  MoveL 668 to (230.14, 163.68, 22.22) mm, rotated rx 180 ry 0 rz -160 deg; joints [-25.106, 26.658, 31.364, 9.576, 32.341, -8.112]
  Call Extruder(552.80049)
  MoveL 669 to (229.91, 163.75, 22.22) mm, rotated rx 180 ry 0 rz -180 deg; joints [-30.703, 36.195, 15.324, 43.661, 47.695, -32.714]
  MoveL 670 to (229.91, 163.75, 22.22) mm, rotated rx -180 ry 0 rz 180 deg; joints [-30.703, 36.195, 15.324, 43.661, 47.695, -32.714]
  Call Extruder(553.06879)
  MoveL 671 to (229.69, 163.82, 22.23) mm, rotated rx 180 ry 0 rz 180 deg; joints [-30.721, 35.901, 15.858, 43.833, 47.531, -32.953]
  MoveL 672 to (229.69, 163.82, 22.23) mm, rotated rx 180 ry 0 rz 180 deg; joints [-30.721, 35.901, 15.858, 43.833, 47.531, -32.953]
  Call Extruder(553.30777)
  MoveL 673 to (229.48, 163.86, 22.23) mm, rotated rx 180 ry 0 rz 180 deg; joints [-30.736, 35.656, 16.302, 43.977, 47.396, -33.151]
  MoveL 674 to (229.48, 163.86, 22.23) mm, rotated rx 180 ry 0 rz 180 deg; joints [-30.736, 35.656, 16.302, 43.977, 47.396, -33.151]
  Call Extruder(553.54569)
  MoveL 675 to (229.28, 163.91, 22.22) mm, rotated rx 180 ry 0 rz 180 deg; joints [-30.751, 35.437, 16.698, 44.107, 47.277, -33.33]
  MoveL 676 to (229.28, 163.91, 22.22) mm, rotated rx 180 ry 0 rz 180 deg; joints [-30.751, 35.437, 16.698, 44.107, 47.277, -33.33]
  Call Extruder(553.78253)
  MoveL 677 to (229.08, 163.95, 22.23) mm, rotated rx 180 ry 0 rz 180 deg; joints [-30.766, 35.235, 17.061, 44.227, 47.17, -33.494]
  MoveL 678 to (229.08, 163.95, 22.23) mm, rotated rx 180 ry 0 rz 180 deg; joints [-30.766, 35.235, 17.061, 44.227, 47.17, -33.494]
  Call Extruder(554.01831)
  MoveL 679 to (228.87, 164, 22.23) mm, rotated rx 180 ry 0 rz 180 deg; joints [-30.781, 35.047, 17.397, 44.341, 47.072, -33.647]
  MoveL 680 to (228.87, 164, 22.23) mm, rotated rx 180 ry 0 rz 180 deg; joints [-30.781, 35.047, 17.397, 44.341, 47.072, -33.647]
  Call Extruder(554.27820)
  MoveL 681 to (228.64, 164.04, 22.23) mm, rotated rx -180 ry 0 rz -180 deg; joints [-30.797, 34.852, 17.746, 44.459, 46.971, -33.806]
  MoveL 682 to (228.64, 164.04, 22.23) mm, rotated rx -180 ry 0 rz -180 deg; joints [-30.797, 34.852, 17.746, 44.459, 46.971, -33.806]
  Call Extruder(554.56187)
  MoveL 683 to (228.4, 164.09, 22.22) mm, rotated rx 180 ry 0 rz -180 deg; joints [-30.815, 34.649, 18.106, 44.582, 46.869, -33.971]
  MoveL 684 to (228.4, 164.09, 22.22) mm, rotated rx 180 ry 0 rz -180 deg; joints [-30.815, 34.649, 18.106, 44.582, 46.869, -33.971]
  Call Extruder(554.84409)
  MoveL 685 to (228.15, 164.14, 22.22) mm, rotated rx 180 ry 0 rz 180 deg; joints [-30.832, 34.457, 18.446, 44.7, 46.773, -34.128]
  MoveL 686 to (228.15, 164.14, 22.22) mm, rotated rx 180 ry 0 rz 180 deg; joints [-30.832, 34.457, 18.446, 44.7, 46.773, -34.128]
  Call Extruder(555.12487)
  MoveL 687 to (227.9, 164.19, 22.23) mm, rotated rx 180 ry 0 rz 180 deg; joints [-30.85, 34.276, 18.766, 44.812, 46.685, -34.276]
  MoveL 688 to (227.9, 164.19, 22.23) mm, rotated rx 180 ry 0 rz 180 deg; joints [-30.85, 34.276, 18.766, 44.812, 46.685, -34.276]
  Call Extruder(555.40421)
  MoveL 689 to (227.65, 164.24, 22.22) mm, rotated rx 180 ry 0 rz 180 deg; joints [-30.868, 34.103, 19.07, 44.92, 46.602, -34.417]
  MoveL 690 to (227.65, 164.24, 22.22) mm, rotated rx 180 ry 0 rz 180 deg; joints [-30.868, 34.103, 19.07, 44.92, 46.602, -34.417]
  Call Extruder(555.68211)
  MoveL 691 to (227.4, 164.29, 22.23) mm, rotated rx -180 ry 0 rz -180 deg; joints [-30.886, 33.937, 19.361, 45.024, 46.523, -34.552]
  MoveL 692 to (227.4, 164.29, 22.23) mm, rotated rx -180 ry 0 rz -180 deg; joints [-30.886, 33.937, 19.361, 45.024, 46.523, -34.552]
  Call Extruder(555.95856)
  MoveL 693 to (227.15, 164.34, 22.22) mm, rotated rx 180 ry 0 rz 180 deg; joints [-30.903, 33.778, 19.639, 45.124, 46.449, -34.683]
  MoveL 694 to (227.15, 164.34, 22.22) mm, rotated rx 180 ry 0 rz 180 deg; joints [-30.903, 33.778, 19.639, 45.124, 46.449, -34.683]
  Call Extruder(556.26358)
  MoveL 695 to (226.87, 164.39, 22.23) mm, rotated rx 180 ry 0 rz 180 deg; joints [-30.923, 33.605, 19.941, 45.233, 46.369, -34.824]
  MoveL 696 to (226.87, 164.39, 22.23) mm, rotated rx 180 ry 0 rz 180 deg; joints [-30.923, 33.605, 19.941, 45.233, 46.369, -34.824]
  Call Extruder(556.59701)
  MoveL 697 to (226.57, 164.44, 22.22) mm, rotated rx 180 ry 0 rz 180 deg; joints [-30.943, 33.419, 20.264, 45.349, 46.284, -34.975]
  MoveL 698 to (226.57, 164.44, 22.22) mm, rotated rx 180 ry 0 rz 180 deg; joints [-30.943, 33.419, 20.264, 45.349, 46.284, -34.975]
  Call Extruder(556.92871)
  MoveL 699 to (226.26, 164.49, 22.22) mm, rotated rx -180 ry 0 rz 180 deg; joints [-30.964, 33.24, 20.575, 45.463, 46.204, -35.121]
  MoveL 700 to (226.26, 164.49, 22.22) mm, rotated rx -180 ry 0 rz 180 deg; joints [-30.964, 33.24, 20.575, 45.463, 46.204, -35.121]
  Call Extruder(557.25870)
  MoveL 701 to (225.96, 164.54, 22.22) mm, rotated rx 180 ry 0 rz 180 deg; joints [-30.985, 33.068, 20.873, 45.572, 46.128, -35.262]
  MoveL 702 to (225.96, 164.54, 22.22) mm, rotated rx 180 ry 0 rz 180 deg; joints [-30.985, 33.068, 20.873, 45.572, 46.128, -35.262]
  Call Extruder(557.58696)
  MoveL 703 to (225.65, 164.58, 22.22) mm, rotated rx 180 ry 0 rz 180 deg; joints [-31.006, 32.901, 21.16, 45.679, 46.056, -35.397]
  MoveL 704 to (225.65, 164.58, 22.22) mm, rotated rx 180 ry 0 rz 180 deg; joints [-31.006, 32.901, 21.16, 45.679, 46.056, -35.397]
  Call Extruder(557.91351)
  MoveL 705 to (225.34, 164.63, 22.23) mm, rotated rx 180 ry 0 rz 180 deg; joints [-31.027, 32.739, 21.438, 45.783, 45.987, -35.53]
  MoveL 706 to (225.34, 164.63, 22.23) mm, rotated rx 180 ry 0 rz 180 deg; joints [-31.027, 32.739, 21.438, 45.783, 45.987, -35.53]
  Call Extruder(558.28060)
  MoveL 707 to (225, 164.68, 22.23) mm, rotated rx 180 ry 0 rz 180 deg; joints [-31.049, 32.558, 21.749, 45.898, 45.91, -35.677]
  MoveL 708 to (225, 164.68, 22.23) mm, rotated rx 180 ry 0 rz 180 deg; joints [-31.049, 32.558, 21.749, 45.898, 45.91, -35.677]
  Call Extruder(558.68804)
  MoveL 709 to (224.61, 164.73, 22.22) mm, rotated rx 180 ry 0 rz 180 deg; joints [-31.074, 32.36, 22.086, 46.024, 45.827, -35.836]
  MoveL 710 to (224.61, 164.73, 22.22) mm, rotated rx 180 ry 0 rz 180 deg; joints [-31.074, 32.36, 22.086, 46.024, 45.827, -35.836]
  Call Extruder(559.09343)
  MoveL 711 to (224.22, 164.77, 22.22) mm, rotated rx 180 ry 0 rz 180 deg; joints [-31.1, 32.168, 22.413, 46.147, 45.749, -35.991]
  MoveL 712 to (224.22, 164.77, 22.22) mm, rotated rx 180 ry 0 rz 180 deg; joints [-31.1, 32.168, 22.413, 46.147, 45.749, -35.991]
  Call Extruder(559.49678)
  MoveL 713 to (223.84, 164.82, 22.23) mm, rotated rx 180 ry 0 rz 180 deg; joints [-31.125, 31.983, 22.728, 46.266, 45.674, -36.142]
  MoveL 714 to (223.84, 164.82, 22.23) mm, rotated rx 180 ry 0 rz 180 deg; joints [-31.125, 31.983, 22.728, 46.266, 45.674, -36.142]
  Call Extruder(559.89807)
  MoveL 715 to (223.45, 164.86, 22.22) mm, rotated rx 180 ry 0 rz 180 deg; joints [-31.15, 31.801, 23.035, 46.383, 45.602, -36.288]
  MoveL 716 to (223.45, 164.86, 22.22) mm, rotated rx 180 ry 0 rz 180 deg; joints [-31.15, 31.801, 23.035, 46.383, 45.602, -36.288]
  Call Extruder(560.50287)
  MoveL 717 to (222.86, 164.91, 22.22) mm, rotated rx 180 ry 0 rz 180 deg; joints [-31.186, 31.529, 23.494, 46.557, 45.495, -36.506]
  MoveL 718 to (222.86, 164.91, 22.22) mm, rotated rx 180 ry 0 rz 180 deg; joints [-31.186, 31.529, 23.494, 46.557, 45.495, -36.506]
  Call Extruder(561.10453)
  MoveL 719 to (222.27, 164.96, 22.22) mm, rotated rx 180 ry 0 rz -180 deg; joints [-31.222, 31.266, 23.935, 46.725, 45.394, -36.717]
  MoveL 720 to (222.27, 164.96, 22.22) mm, rotated rx 180 ry 0 rz -180 deg; joints [-31.222, 31.266, 23.935, 46.725, 45.394, -36.717]
  Call Extruder(561.70303)
  MoveL 721 to (221.68, 165, 22.22) mm, rotated rx 180 ry 0 rz 180 deg; joints [-31.258, 31.012, 24.358, 46.888, 45.3, -36.92]
  MoveL 722 to (221.68, 165, 22.22) mm, rotated rx 180 ry 0 rz 180 deg; joints [-31.258, 31.012, 24.358, 46.888, 45.3, -36.92]
  Call Extruder(562.87480)
  MoveL 723 to (220.52, 165.05, 22.22) mm, rotated rx 180 ry 0 rz 180 deg; joints [-31.326, 30.522, 25.171, 47.199, 45.12, -37.307]
  MoveL 724 to (220.52, 165.05, 22.22) mm, rotated rx 180 ry 0 rz 180 deg; joints [-31.326, 30.522, 25.171, 47.199, 45.12, -37.307]
  Call Extruder(564.33276)
  MoveL 725 to (219.06, 165.09, 22.23) mm, rotated rx -180 ry 0 rz 180 deg; joints [-31.409, 29.942, 26.126, 47.568, 44.918, -37.762]
  Call Extruder(802.92585)
  MoveL 726 to (-19.06, 165.09, 22.22) mm, rotated rx 180 ry 0 rz 180 deg; joints [-51.475, -6.461, 71.178, 71.221, 55.723, -58.879]
  Call Extruder(803.80103)
  MoveL 727 to (-19.94, 165.07, 22.23) mm, rotated rx 180 ry 0 rz 180 deg; joints [-51.582, -6.542, 71.249, 71.281, 55.818, -58.905]
  MoveL 728 to (-19.94, 165.07, 22.23) mm, rotated rx 180 ry 0 rz 180 deg; joints [-51.582, -6.542, 71.249, 71.281, 55.818, -58.905]
  Call Extruder(804.97281)
  MoveL 729 to (-21.1, 165.03, 22.22) mm, rotated rx -180 ry 0 rz -180 deg; joints [-51.722, -6.651, 71.345, 71.36, 55.943, -58.938]
  MoveL 730 to (-21.1, 165.03, 22.22) mm, rotated rx -180 ry 0 rz -180 deg; joints [-51.722, -6.651, 71.345, 71.36, 55.943, -58.938]
  Call Extruder(805.86087)
  MoveL 731 to (-21.97, 164.98, 22.22) mm, rotated rx 180 ry 0 rz 180 deg; joints [-51.827, -6.735, 71.417, 71.418, 56.036, -58.962]
  MoveL 732 to (-21.97, 164.98, 22.22) mm, rotated rx 180 ry 0 rz 180 deg; joints [-51.827, -6.735, 71.417, 71.418, 56.036, -58.962]
  Call Extruder(806.46253)
  MoveL 733 to (-22.56, 164.93, 22.22) mm, rotated rx 180 ry 0 rz 180 deg; joints [-51.897, -6.793, 71.468, 71.456, 56.098, -58.977]
  MoveL 734 to (-22.56, 164.93, 22.22) mm, rotated rx 180 ry 0 rz 180 deg; joints [-51.897, -6.793, 71.468, 71.456, 56.098, -58.977]
  Call Extruder(807.06734)
  MoveL 735 to (-23.15, 164.89, 22.22) mm, rotated rx -180 ry 0 rz 180 deg; joints [-51.966, -6.851, 71.518, 71.494, 56.16, -58.993]
  MoveL 736 to (-23.15, 164.89, 22.22) mm, rotated rx -180 ry 0 rz 180 deg; joints [-51.966, -6.851, 71.518, 71.494, 56.16, -58.993]
  Call Extruder(807.57186)
  MoveL 737 to (-23.64, 164.84, 22.22) mm, rotated rx 180 ry 0 rz 180 deg; joints [-52.023, -6.9, 71.56, 71.525, 56.211, -59.005]
  MoveL 738 to (-23.64, 164.84, 22.22) mm, rotated rx 180 ry 0 rz 180 deg; joints [-52.023, -6.9, 71.56, 71.525, 56.211, -59.005]
  Call Extruder(807.97520)
  MoveL 739 to (-24.03, 164.79, 22.22) mm, rotated rx 180 ry 0 rz 180 deg; joints [-52.067, -6.939, 71.595, 71.55, 56.25, -59.014]
  MoveL 740 to (-24.03, 164.79, 22.22) mm, rotated rx 180 ry 0 rz 180 deg; joints [-52.067, -6.939, 71.595, 71.55, 56.25, -59.014]
  Call Extruder(808.38059)
  MoveL 741 to (-24.42, 164.75, 22.22) mm, rotated rx 180 ry 0 rz 180 deg; joints [-52.112, -6.979, 71.629, 71.574, 56.29, -59.023]
  MoveL 742 to (-24.42, 164.75, 22.22) mm, rotated rx 180 ry 0 rz 180 deg; joints [-52.112, -6.979, 71.629, 71.574, 56.29, -59.023]
  Call Extruder(808.78804)
  MoveL 743 to (-24.8, 164.7, 22.23) mm, rotated rx 180 ry 0 rz 180 deg; joints [-52.156, -7.019, 71.663, 71.598, 56.33, -59.032]
  MoveL 744 to (-24.8, 164.7, 22.23) mm, rotated rx 180 ry 0 rz 180 deg; joints [-52.156, -7.019, 71.663, 71.598, 56.33, -59.032]
  Call Extruder(809.19753)
  MoveL 745 to (-25.19, 164.66, 22.22) mm, rotated rx 180 ry 0 rz -180 deg; joints [-52.2, -7.058, 71.697, 71.622, 56.37, -59.041]
  MoveL 746 to (-25.19, 164.66, 22.22) mm, rotated rx 180 ry 0 rz -180 deg; joints [-52.2, -7.058, 71.697, 71.622, 56.37, -59.041]
  Call Extruder(809.52408)
  MoveL 747 to (-25.5, 164.61, 22.22) mm, rotated rx 180 ry 0 rz 180 deg; joints [-52.235, -7.091, 71.725, 71.64, 56.4, -59.048]
  MoveL 748 to (-25.5, 164.61, 22.22) mm, rotated rx 180 ry 0 rz 180 deg; joints [-52.235, -7.091, 71.725, 71.64, 56.4, -59.048]
  Call Extruder(809.85235)
  MoveL 749 to (-25.8, 164.56, 22.22) mm, rotated rx 180 ry 0 rz 180 deg; joints [-52.269, -7.123, 71.753, 71.658, 56.431, -59.054]
  MoveL 750 to (-25.8, 164.56, 22.22) mm, rotated rx 180 ry 0 rz 180 deg; joints [-52.269, -7.123, 71.753, 71.658, 56.431, -59.054]
  Call Extruder(810.18235)
  MoveL 751 to (-26.11, 164.51, 22.22) mm, rotated rx 180 ry 0 rz -180 deg; joints [-52.303, -7.156, 71.781, 71.676, 56.461, -59.061]
  MoveL 752 to (-26.11, 164.51, 22.22) mm, rotated rx 180 ry 0 rz -180 deg; joints [-52.303, -7.156, 71.781, 71.676, 56.461, -59.061]
  Call Extruder(810.51406)
  MoveL 753 to (-26.41, 164.46, 22.22) mm, rotated rx -180 ry 0 rz 180 deg; joints [-52.337, -7.188, 71.809, 71.695, 56.492, -59.067]
  MoveL 754 to (-26.41, 164.46, 22.22) mm, rotated rx -180 ry 0 rz 180 deg; joints [-52.337, -7.188, 71.809, 71.695, 56.492, -59.067]
  Call Extruder(810.84750)
  MoveL 755 to (-26.72, 164.41, 22.22) mm, rotated rx 180 ry 0 rz 180 deg; joints [-52.371, -7.221, 71.837, 71.713, 56.523, -59.074]
  MoveL 756 to (-26.72, 164.41, 22.22) mm, rotated rx 180 ry 0 rz 180 deg; joints [-52.371, -7.221, 71.837, 71.713, 56.523, -59.074]
  Call Extruder(811.18265)
  MoveL 757 to (-27.03, 164.37, 22.22) mm, rotated rx 180 ry 0 rz 180 deg; joints [-52.405, -7.253, 71.865, 71.731, 56.554, -59.08]
  MoveL 758 to (-27.03, 164.37, 22.22) mm, rotated rx 180 ry 0 rz 180 deg; joints [-52.405, -7.253, 71.865, 71.731, 56.554, -59.08]
  Call Extruder(811.45910)
  MoveL 759 to (-27.27, 164.32, 22.22) mm, rotated rx 180 ry 0 rz 180 deg; joints [-52.432, -7.28, 71.889, 71.745, 56.578, -59.085]
  MoveL 760 to (-27.27, 164.32, 22.22) mm, rotated rx 180 ry 0 rz 180 deg; joints [-52.432, -7.28, 71.889, 71.745, 56.578, -59.085]
  Call Extruder(811.73700)
  MoveL 761 to (-27.52, 164.27, 22.22) mm, rotated rx 180 ry 0 rz 180 deg; joints [-52.459, -7.308, 71.912, 71.759, 56.602, -59.09]
  MoveL 762 to (-27.52, 164.27, 22.22) mm, rotated rx 180 ry 0 rz 180 deg; joints [-52.459, -7.308, 71.912, 71.759, 56.602, -59.09]
  Call Extruder(812.01634)
  MoveL 763 to (-27.77, 164.22, 22.23) mm, rotated rx -180 ry 0 rz 180 deg; joints [-52.486, -7.336, 71.936, 71.773, 56.626, -59.094]
  MoveL 764 to (-27.77, 164.22, 22.23) mm, rotated rx -180 ry 0 rz 180 deg; joints [-52.486, -7.336, 71.936, 71.773, 56.626, -59.094]
  Call Extruder(812.29712)
  MoveL 765 to (-28.02, 164.17, 22.22) mm, rotated rx 180 ry 0 rz -180 deg; joints [-52.513, -7.363, 71.959, 71.787, 56.651, -59.099]
  MoveL 766 to (-28.02, 164.17, 22.22) mm, rotated rx 180 ry 0 rz -180 deg; joints [-52.513, -7.363, 71.959, 71.787, 56.651, -59.099]
  Call Extruder(812.57934)
  MoveL 767 to (-28.27, 164.12, 22.22) mm, rotated rx 180 ry 0 rz 180 deg; joints [-52.54, -7.39, 71.983, 71.802, 56.675, -59.104]
  MoveL 768 to (-28.27, 164.12, 22.22) mm, rotated rx 180 ry 0 rz 180 deg; joints [-52.54, -7.39, 71.983, 71.802, 56.675, -59.104]
  Call Extruder(812.75508)
  MoveL 769 to (-28.43, 164.09, 22.22) mm, rotated rx -180 ry 0 rz 180 deg; joints [-52.556, -7.407, 71.997, 71.81, 56.69, -59.107]
  Set speed (130.0 mm/s)
  MoveL 770 to (-31.76, 163.31, 22.22) mm, rotated rx -180 ry 0 rz 180 deg; joints [-52.91, -7.786, 72.32, 71.992, 57.011, -59.161]
  MoveL 771 to (-31.76, 163.31, 31.63) mm, rotated rx 180 ry 0 rz 180 deg; joints [-52.91, -8.807, 74.811, 72.909, 56.568, -60.836]
  Call Extruder(810.75508)
  Set speed (40.0 mm/s)
  MoveL 772 to (-31.76, 163.31, 31.63) mm, rotated rx 180 ry 0 rz 180 deg; joints [-52.91, -8.807, 74.811, 72.909, 56.568, -60.836]
  Call Extruder(0.00000)
  Set speed (130.0 mm/s)
  MoveL 773 to (-39.41, 155.44, 31.63) mm, rotated rx 180 ry 0 rz 180 deg; joints [-53.137, -10.347, 76.07, 72.866, 56.849, -60.587]
  Call Extruder(2.00000)
  Set speed (40.0 mm/s)
  MoveL 774 to (-39.41, 155.44, 31.63) mm, rotated rx 180 ry 0 rz 180 deg; joints [-53.137, -10.347, 76.07, 72.866, 56.849, -60.587]
  Set speed (30.0 mm/s)
  MoveL 775 to (-39.41, 155.44, 31.63) mm, rotated rx 180 ry 0 rz 180 deg; joints [-53.137, -10.347, 76.07, 72.866, 56.849, -60.587]
  Call Extruder(2.11346)
  MoveL 776 to (-39.47, 155.25, 31.63) mm, rotated rx 180 ry 0 rz 180 deg; joints [-53.126, -10.374, 76.091, 72.856, 56.841, -60.578]
  MoveL 777 to (-39.47, 155.25, 31.63) mm, rotated rx 180 ry 0 rz 180 deg; joints [-53.126, -10.374, 76.091, 72.856, 56.841, -60.578]
  Call Extruder(2.22647)
  MoveL 778 to (-39.53, 155.06, 31.63) mm, rotated rx -180 ry 0 rz 180 deg; joints [-53.115, -10.4, 76.112, 72.847, 56.833, -60.568]
  MoveL 779 to (-39.53, 155.06, 31.63) mm, rotated rx -180 ry 0 rz 180 deg; joints [-53.115, -10.4, 76.112, 72.847, 56.833, -60.568]
  Call Extruder(2.33904)
  MoveL 780 to (-39.59, 154.87, 31.63) mm, rotated rx 180 ry 0 rz -180 deg; joints [-53.105, -10.426, 76.133, 72.837, 56.825, -60.559]
  MoveL 781 to (-39.59, 154.87, 31.63) mm, rotated rx 180 ry 0 rz -180 deg; joints [-53.105, -10.426, 76.133, 72.837, 56.825, -60.559]
  Call Extruder(2.45116)
  MoveL 782 to (-39.65, 154.68, 31.63) mm, rotated rx 180 ry 0 rz 180 deg; joints [-53.094, -10.453, 76.154, 72.827, 56.817, -60.55]
  MoveL 783 to (-39.65, 154.68, 31.63) mm, rotated rx 180 ry 0 rz 180 deg; joints [-53.094, -10.453, 76.154, 72.827, 56.817, -60.55]
  Call Extruder(2.56284)
  MoveL 784 to (-39.71, 154.5, 31.63) mm, rotated rx 180 ry 0 rz -180 deg; joints [-53.083, -10.479, 76.175, 72.818, 56.809, -60.54]
  MoveL 785 to (-39.71, 154.5, 31.63) mm, rotated rx 180 ry 0 rz -180 deg; joints [-53.083, -10.479, 76.175, 72.818, 56.809, -60.54]
  Call Extruder(2.69391)
  MoveL 786 to (-39.78, 154.27, 31.63) mm, rotated rx 180 ry 0 rz 180 deg; joints [-53.069, -10.51, 76.2, 72.806, 56.8, -60.529]
  MoveL 787 to (-39.78, 154.27, 31.63) mm, rotated rx 180 ry 0 rz 180 deg; joints [-53.069, -10.51, 76.2, 72.806, 56.8, -60.529]
  Call Extruder(2.82442)
  MoveL 788 to (-39.85, 154.05, 31.63) mm, rotated rx 180 ry 0 rz -180 deg; joints [-53.056, -10.54, 76.224, 72.794, 56.79, -60.517]
  MoveL 789 to (-39.85, 154.05, 31.63) mm, rotated rx 180 ry 0 rz -180 deg; joints [-53.056, -10.54, 76.224, 72.794, 56.79, -60.517]
  Call Extruder(2.95437)
  MoveL 790 to (-39.92, 153.82, 31.63) mm, rotated rx 180 ry 0 rz -180 deg; joints [-53.042, -10.571, 76.249, 72.782, 56.78, -60.506]
  MoveL 791 to (-39.92, 153.82, 31.63) mm, rotated rx 180 ry 0 rz -180 deg; joints [-53.042, -10.571, 76.249, 72.782, 56.78, -60.506]
  Call Extruder(3.08375)
  MoveL 792 to (-39.98, 153.6, 31.63) mm, rotated rx 180 ry 0 rz 180 deg; joints [-53.029, -10.602, 76.273, 72.77, 56.77, -60.494]
  MoveL 793 to (-39.98, 153.6, 31.63) mm, rotated rx 180 ry 0 rz 180 deg; joints [-53.029, -10.602, 76.273, 72.77, 56.77, -60.494]
  Call Extruder(3.20572)
  MoveL 794 to (-40.04, 153.39, 31.63) mm, rotated rx 180 ry 0 rz 180 deg; joints [-53.015, -10.631, 76.296, 72.758, 56.759, -60.483]
  MoveL 795 to (-40.04, 153.39, 31.63) mm, rotated rx 180 ry 0 rz 180 deg; joints [-53.015, -10.631, 76.296, 72.758, 56.759, -60.483]
  Call Extruder(3.32058)
  MoveL 796 to (-40.08, 153.18, 31.63) mm, rotated rx 180 ry 0 rz 180 deg; joints [-53, -10.657, 76.317, 72.746, 56.748, -60.472]
  MoveL 797 to (-40.08, 153.18, 31.63) mm, rotated rx 180 ry 0 rz 180 deg; joints [-53, -10.657, 76.317, 72.746, 56.748, -60.472]
  Call Extruder(3.43499)
  MoveL 798 to (-40.13, 152.98, 31.63) mm, rotated rx 180 ry 0 rz 180 deg; joints [-52.985, -10.684, 76.338, 72.734, 56.737, -60.461]
  MoveL 799 to (-40.13, 152.98, 31.63) mm, rotated rx 180 ry 0 rz 180 deg; joints [-52.985, -10.684, 76.338, 72.734, 56.737, -60.461]
  Call Extruder(3.54895)
  MoveL 800 to (-40.17, 152.77, 31.63) mm, rotated rx -180 ry 0 rz 180 deg; joints [-52.97, -10.71, 76.36, 72.722, 56.725, -60.45]
  MoveL 801 to (-40.17, 152.77, 31.63) mm, rotated rx -180 ry 0 rz 180 deg; joints [-52.97, -10.71, 76.36, 72.722, 56.725, -60.45]
  Call Extruder(3.66245)
  MoveL 802 to (-40.22, 152.57, 31.63) mm, rotated rx 180 ry 0 rz 180 deg; joints [-52.956, -10.737, 76.381, 72.71, 56.714, -60.439]
  MoveL 803 to (-40.22, 152.57, 31.63) mm, rotated rx 180 ry 0 rz 180 deg; joints [-52.956, -10.737, 76.381, 72.71, 56.714, -60.439]
  Call Extruder(3.79973)
  MoveL 804 to (-40.27, 152.32, 31.63) mm, rotated rx -180 ry 0 rz 180 deg; joints [-52.937, -10.769, 76.406, 72.695, 56.7, -60.426]
  MoveL 805 to (-40.27, 152.32, 31.63) mm, rotated rx -180 ry 0 rz 180 deg; joints [-52.937, -10.769, 76.406, 72.695, 56.7, -60.426]
  Call Extruder(3.93640)
  MoveL 806 to (-40.32, 152.07, 31.63) mm, rotated rx -180 ry 0 rz 180 deg; joints [-52.918, -10.801, 76.431, 72.68, 56.686, -60.412]
  MoveL 807 to (-40.32, 152.07, 31.63) mm, rotated rx -180 ry 0 rz 180 deg; joints [-52.918, -10.801, 76.431, 72.68, 56.686, -60.412]
  Call Extruder(4.07246)
  MoveL 808 to (-40.37, 151.82, 31.63) mm, rotated rx 180 ry 0 rz -180 deg; joints [-52.9, -10.833, 76.457, 72.665, 56.671, -60.399]
  MoveL 809 to (-40.37, 151.82, 31.63) mm, rotated rx 180 ry 0 rz -180 deg; joints [-52.9, -10.833, 76.457, 72.665, 56.671, -60.399]
  Call Extruder(4.20791)
  MoveL 810 to (-40.42, 151.57, 31.63) mm, rotated rx 180 ry 0 rz 180 deg; joints [-52.881, -10.865, 76.482, 72.649, 56.657, -60.385]
  MoveL 811 to (-40.42, 151.57, 31.63) mm, rotated rx 180 ry 0 rz 180 deg; joints [-52.881, -10.865, 76.482, 72.649, 56.657, -60.385]
  Call Extruder(4.34275)
  MoveL 812 to (-40.47, 151.32, 31.63) mm, rotated rx 180 ry 0 rz 180 deg; joints [-52.862, -10.897, 76.507, 72.634, 56.643, -60.371]
  MoveL 813 to (-40.47, 151.32, 31.63) mm, rotated rx 180 ry 0 rz 180 deg; joints [-52.862, -10.897, 76.507, 72.634, 56.643, -60.371]
  Call Extruder(4.47698)
  MoveL 814 to (-40.52, 151.07, 31.63) mm, rotated rx 180 ry 0 rz 180 deg; joints [-52.843, -10.928, 76.533, 72.619, 56.628, -60.358]
  MoveL 815 to (-40.52, 151.07, 31.63) mm, rotated rx 180 ry 0 rz 180 deg; joints [-52.843, -10.928, 76.533, 72.619, 56.628, -60.358]
  Call Extruder(4.61060)
  MoveL 816 to (-40.56, 150.83, 31.63) mm, rotated rx 180 ry 0 rz 180 deg; joints [-52.824, -10.96, 76.558, 72.603, 56.614, -60.344]
  MoveL 817 to (-40.56, 150.83, 31.63) mm, rotated rx 180 ry 0 rz 180 deg; joints [-52.824, -10.96, 76.558, 72.603, 56.614, -60.344]
  Call Extruder(4.77270)
  MoveL 818 to (-40.61, 150.52, 31.63) mm, rotated rx 180 ry 0 rz 180 deg; joints [-52.799, -10.998, 76.588, 72.584, 56.595, -60.327]
  MoveL 819 to (-40.61, 150.52, 31.63) mm, rotated rx 180 ry 0 rz 180 deg; joints [-52.799, -10.998, 76.588, 72.584, 56.595, -60.327]
  Call Extruder(4.93406)
  MoveL 820 to (-40.66, 150.21, 31.63) mm, rotated rx 180 ry 0 rz 180 deg; joints [-52.775, -11.037, 76.618, 72.564, 56.575, -60.309]
  MoveL 821 to (-40.66, 150.21, 31.63) mm, rotated rx 180 ry 0 rz 180 deg; joints [-52.775, -11.037, 76.618, 72.564, 56.575, -60.309]
  Call Extruder(5.09469)
  MoveL 822 to (-40.71, 149.91, 31.63) mm, rotated rx -180 ry 0 rz 180 deg; joints [-52.75, -11.075, 76.648, 72.544, 56.556, -60.292]
  MoveL 823 to (-40.71, 149.91, 31.63) mm, rotated rx -180 ry 0 rz 180 deg; joints [-52.75, -11.075, 76.648, 72.544, 56.556, -60.292]
  Call Extruder(5.25460)
  MoveL 824 to (-40.76, 149.6, 31.63) mm, rotated rx -180 ry 0 rz 180 deg; joints [-52.725, -11.113, 76.678, 72.524, 56.537, -60.275]
  MoveL 825 to (-40.76, 149.6, 31.63) mm, rotated rx -180 ry 0 rz 180 deg; joints [-52.725, -11.113, 76.678, 72.524, 56.537, -60.275]
  Call Extruder(5.41378)
  MoveL 826 to (-40.81, 149.3, 31.63) mm, rotated rx -180 ry 0 rz 180 deg; joints [-52.7, -11.151, 76.708, 72.504, 56.518, -60.257]
  MoveL 827 to (-40.81, 149.3, 31.63) mm, rotated rx -180 ry 0 rz 180 deg; joints [-52.7, -11.151, 76.708, 72.504, 56.518, -60.257]
  Call Extruder(5.57223)
  MoveL 828 to (-40.86, 148.99, 31.63) mm, rotated rx 180 ry 0 rz 180 deg; joints [-52.675, -11.189, 76.738, 72.484, 56.498, -60.24]
  MoveL 829 to (-40.86, 148.99, 31.63) mm, rotated rx 180 ry 0 rz 180 deg; joints [-52.675, -11.189, 76.738, 72.484, 56.498, -60.24]
  Call Extruder(5.77111)
  MoveL 830 to (-40.9, 148.6, 31.63) mm, rotated rx 180 ry 0 rz 180 deg; joints [-52.641, -11.235, 76.775, 72.458, 56.472, -60.217]
  MoveL 831 to (-40.9, 148.6, 31.63) mm, rotated rx 180 ry 0 rz 180 deg; joints [-52.641, -11.235, 76.775, 72.458, 56.472, -60.217]
  Call Extruder(5.96911)
  MoveL 832 to (-40.95, 148.22, 31.63) mm, rotated rx -180 ry 0 rz 180 deg; joints [-52.607, -11.282, 76.811, 72.431, 56.445, -60.194]
  MoveL 833 to (-40.95, 148.22, 31.63) mm, rotated rx -180 ry 0 rz 180 deg; joints [-52.607, -11.282, 76.811, 72.431, 56.445, -60.194]
  Call Extruder(6.16625)
  MoveL 834 to (-40.99, 147.83, 31.63) mm, rotated rx 180 ry 0 rz -180 deg; joints [-52.573, -11.329, 76.848, 72.404, 56.419, -60.172]
  MoveL 835 to (-40.99, 147.83, 31.63) mm, rotated rx 180 ry 0 rz -180 deg; joints [-52.573, -11.329, 76.848, 72.404, 56.419, -60.172]
  Call Extruder(6.36252)
  MoveL 836 to (-41.04, 147.44, 31.63) mm, rotated rx 180 ry 0 rz 180 deg; joints [-52.539, -11.375, 76.884, 72.377, 56.392, -60.149]
  MoveL 837 to (-41.04, 147.44, 31.63) mm, rotated rx 180 ry 0 rz 180 deg; joints [-52.539, -11.375, 76.884, 72.377, 56.392, -60.149]
  Call Extruder(6.60821)
  MoveL 838 to (-41.09, 146.95, 31.63) mm, rotated rx 180 ry 0 rz 180 deg; joints [-52.494, -11.433, 76.93, 72.343, 56.357, -60.12]
  MoveL 839 to (-41.09, 146.95, 31.63) mm, rotated rx 180 ry 0 rz 180 deg; joints [-52.494, -11.433, 76.93, 72.343, 56.357, -60.12]
  Call Extruder(6.90294)
  MoveL 840 to (-41.13, 146.36, 31.63) mm, rotated rx 180 ry 0 rz -180 deg; joints [-52.439, -11.502, 76.983, 72.3, 56.314, -60.084]
  MoveL 841 to (-41.13, 146.36, 31.63) mm, rotated rx 180 ry 0 rz -180 deg; joints [-52.439, -11.502, 76.983, 72.3, 56.314, -60.084]
  Call Extruder(7.19634)
  MoveL 842 to (-41.18, 145.77, 31.63) mm, rotated rx 180 ry 0 rz 180 deg; joints [-52.383, -11.571, 77.037, 72.257, 56.27, -60.048]
  MoveL 843 to (-41.18, 145.77, 31.63) mm, rotated rx 180 ry 0 rz 180 deg; joints [-52.383, -11.571, 77.037, 72.257, 56.27, -60.048]
  Call Extruder(7.62967)
  MoveL 844 to (-41.22, 144.9, 31.63) mm, rotated rx -180 ry 0 rz 180 deg; joints [-52.297, -11.671, 77.115, 72.191, 56.203, -59.994]
  MoveL 845 to (-41.22, 144.9, 31.63) mm, rotated rx -180 ry 0 rz 180 deg; joints [-52.297, -11.671, 77.115, 72.191, 56.203, -59.994]
  Call Extruder(8.20183)
  MoveL 846 to (-41.27, 143.74, 31.63) mm, rotated rx 180 ry 0 rz -180 deg; joints [-52.18, -11.802, 77.217, 72.102, 56.111, -59.921]
  MoveL 847 to (-41.27, 143.74, 31.63) mm, rotated rx 180 ry 0 rz -180 deg; joints [-52.18, -11.802, 77.217, 72.102, 56.111, -59.921]
  Call Extruder(8.62966)
  MoveL 848 to (-41.29, 142.86, 31.63) mm, rotated rx 180 ry 0 rz 180 deg; joints [-52.09, -11.899, 77.292, 72.033, 56.039, -59.865]
  Call Extruder(50.62319)
  MoveL 849 to (-41.29, 57.14, 31.63) mm, rotated rx 180 ry 0 rz 180 deg; joints [-40.759, -20.206, 83.021, 62.074, 47.639, -51.809]
  MoveL 850 to (-41.29, 57.14, 31.63) mm, rotated rx 180 ry 0 rz 180 deg; joints [-40.759, -20.206, 83.021, 62.074, 47.639, -51.809]
  Call Extruder(51.33876)
  MoveL 851 to (-41.25, 55.68, 31.63) mm, rotated rx -180 ry 0 rz 180 deg; joints [-40.517, -20.323, 83.092, 61.833, 47.471, -51.616]
  MoveL 852 to (-41.25, 55.68, 31.63) mm, rotated rx -180 ry 0 rz 180 deg; joints [-40.517, -20.323, 83.092, 61.833, 47.471, -51.616]
  Call Extruder(51.91350)
  MoveL 853 to (-41.2, 54.52, 31.63) mm, rotated rx 180 ry 0 rz 180 deg; joints [-40.32, -20.415, 83.147, 61.638, 47.335, -51.46]
  MoveL 854 to (-41.2, 54.52, 31.63) mm, rotated rx 180 ry 0 rz 180 deg; joints [-40.32, -20.415, 83.147, 61.638, 47.335, -51.46]
  Call Extruder(52.20690)
  MoveL 855 to (-41.15, 53.93, 31.63) mm, rotated rx 180 ry 0 rz 180 deg; joints [-40.217, -20.459, 83.174, 61.536, 47.263, -51.379]
  MoveL 856 to (-41.15, 53.93, 31.63) mm, rotated rx 180 ry 0 rz 180 deg; joints [-40.217, -20.459, 83.174, 61.536, 47.263, -51.379]
  Call Extruder(52.50163)
  MoveL 857 to (-41.11, 53.34, 31.63) mm, rotated rx 180 ry 0 rz 180 deg; joints [-40.114, -20.503, 83.2, 61.433, 47.19, -51.299]
  MoveL 858 to (-41.11, 53.34, 31.63) mm, rotated rx 180 ry 0 rz 180 deg; joints [-40.114, -20.503, 83.2, 61.433, 47.19, -51.299]
  Call Extruder(52.79770)
  MoveL 859 to (-41.06, 52.75, 31.63) mm, rotated rx -180 ry 0 rz 180 deg; joints [-40.01, -20.547, 83.226, 61.33, 47.118, -51.217]
  MoveL 860 to (-41.06, 52.75, 31.63) mm, rotated rx -180 ry 0 rz 180 deg; joints [-40.01, -20.547, 83.226, 61.33, 47.118, -51.217]
  Call Extruder(52.99397)
  MoveL 861 to (-41.02, 52.37, 31.63) mm, rotated rx 180 ry 0 rz 180 deg; joints [-39.939, -20.575, 83.243, 61.261, 47.068, -51.163]
  MoveL 862 to (-41.02, 52.37, 31.63) mm, rotated rx 180 ry 0 rz 180 deg; joints [-39.939, -20.575, 83.243, 61.261, 47.068, -51.163]
  Call Extruder(53.19111)
  MoveL 863 to (-40.97, 51.98, 31.63) mm, rotated rx 180 ry 0 rz 180 deg; joints [-39.869, -20.602, 83.259, 61.192, 47.018, -51.108]
  MoveL 864 to (-40.97, 51.98, 31.63) mm, rotated rx 180 ry 0 rz 180 deg; joints [-39.869, -20.602, 83.259, 61.192, 47.018, -51.108]
  Call Extruder(53.38912)
  MoveL 865 to (-40.92, 51.59, 31.63) mm, rotated rx -180 ry 0 rz 180 deg; joints [-39.798, -20.629, 83.275, 61.122, 46.969, -51.054]
  MoveL 866 to (-40.92, 51.59, 31.63) mm, rotated rx -180 ry 0 rz 180 deg; joints [-39.798, -20.629, 83.275, 61.122, 46.969, -51.054]
  Call Extruder(53.58800)
  MoveL 867 to (-40.88, 51.2, 31.63) mm, rotated rx -180 ry 0 rz 180 deg; joints [-39.727, -20.656, 83.291, 61.052, 46.919, -50.999]
  MoveL 868 to (-40.88, 51.2, 31.63) mm, rotated rx -180 ry 0 rz 180 deg; joints [-39.727, -20.656, 83.291, 61.052, 46.919, -50.999]
  Call Extruder(53.76707)
  MoveL 869 to (-40.83, 50.86, 31.63) mm, rotated rx 180 ry 0 rz 180 deg; joints [-39.663, -20.68, 83.305, 60.989, 46.874, -50.95]
  MoveL 870 to (-40.83, 50.86, 31.63) mm, rotated rx 180 ry 0 rz 180 deg; joints [-39.663, -20.68, 83.305, 60.989, 46.874, -50.95]
  Call Extruder(53.92625)
  MoveL 871 to (-40.78, 50.55, 31.63) mm, rotated rx -180 ry 0 rz 180 deg; joints [-39.605, -20.7, 83.317, 60.932, 46.833, -50.906]
  MoveL 872 to (-40.78, 50.55, 31.63) mm, rotated rx -180 ry 0 rz 180 deg; joints [-39.605, -20.7, 83.317, 60.932, 46.833, -50.906]
  Call Extruder(54.08615)
  MoveL 873 to (-40.74, 50.24, 31.63) mm, rotated rx -180 ry 0 rz 180 deg; joints [-39.547, -20.72, 83.329, 60.875, 46.792, -50.862]
  MoveL 874 to (-40.74, 50.24, 31.63) mm, rotated rx -180 ry 0 rz 180 deg; joints [-39.547, -20.72, 83.329, 60.875, 46.792, -50.862]
  Call Extruder(54.24679)
  MoveL 875 to (-40.69, 49.94, 31.63) mm, rotated rx 180 ry 0 rz 180 deg; joints [-39.489, -20.74, 83.341, 60.819, 46.751, -50.818]
  MoveL 876 to (-40.69, 49.94, 31.63) mm, rotated rx 180 ry 0 rz 180 deg; joints [-39.489, -20.74, 83.341, 60.819, 46.751, -50.818]
  Call Extruder(54.40815)
  MoveL 877 to (-40.64, 49.63, 31.63) mm, rotated rx 180 ry 0 rz 180 deg; joints [-39.431, -20.76, 83.353, 60.762, 46.71, -50.774]
  MoveL 878 to (-40.64, 49.63, 31.63) mm, rotated rx 180 ry 0 rz 180 deg; joints [-39.431, -20.76, 83.353, 60.762, 46.71, -50.774]
  Call Extruder(54.57024)
  MoveL 879 to (-40.59, 49.33, 31.63) mm, rotated rx -180 ry 0 rz 180 deg; joints [-39.373, -20.78, 83.365, 60.704, 46.669, -50.729]
  MoveL 880 to (-40.59, 49.33, 31.63) mm, rotated rx -180 ry 0 rz 180 deg; joints [-39.373, -20.78, 83.365, 60.704, 46.669, -50.729]
  Call Extruder(54.71843)
  MoveL 881 to (-40.54, 49.05, 31.63) mm, rotated rx -180 ry 0 rz 180 deg; joints [-39.32, -20.797, 83.375, 60.652, 46.631, -50.689]
  MoveL 882 to (-40.54, 49.05, 31.63) mm, rotated rx -180 ry 0 rz 180 deg; joints [-39.32, -20.797, 83.375, 60.652, 46.631, -50.689]
  Call Extruder(54.85266)
  MoveL 883 to (-40.49, 48.8, 31.63) mm, rotated rx 180 ry 0 rz 180 deg; joints [-39.271, -20.813, 83.384, 60.604, 46.597, -50.652]
  MoveL 884 to (-40.49, 48.8, 31.63) mm, rotated rx 180 ry 0 rz 180 deg; joints [-39.271, -20.813, 83.384, 60.604, 46.597, -50.652]
  Call Extruder(54.98750)
  MoveL 885 to (-40.44, 48.55, 31.63) mm, rotated rx 180 ry 0 rz 180 deg; joints [-39.222, -20.828, 83.393, 60.557, 46.562, -50.615]
  MoveL 886 to (-40.44, 48.55, 31.63) mm, rotated rx 180 ry 0 rz 180 deg; joints [-39.222, -20.828, 83.393, 60.557, 46.562, -50.615]
  Call Extruder(55.12295)
  MoveL 887 to (-40.39, 48.3, 31.63) mm, rotated rx 180 ry 0 rz -180 deg; joints [-39.174, -20.843, 83.402, 60.509, 46.527, -50.579]
  MoveL 888 to (-40.39, 48.3, 31.63) mm, rotated rx 180 ry 0 rz -180 deg; joints [-39.174, -20.843, 83.402, 60.509, 46.527, -50.579]
  Call Extruder(55.25901)
  MoveL 889 to (-40.34, 48.05, 31.63) mm, rotated rx -180 ry 0 rz 180 deg; joints [-39.125, -20.858, 83.411, 60.461, 46.492, -50.542]
  MoveL 890 to (-40.34, 48.05, 31.63) mm, rotated rx -180 ry 0 rz 180 deg; joints [-39.125, -20.858, 83.411, 60.461, 46.492, -50.542]
  Call Extruder(55.39568)
  MoveL 891 to (-40.29, 47.8, 31.63) mm, rotated rx 180 ry 0 rz -180 deg; joints [-39.076, -20.873, 83.42, 60.413, 46.458, -50.505]
  MoveL 892 to (-40.29, 47.8, 31.63) mm, rotated rx 180 ry 0 rz -180 deg; joints [-39.076, -20.873, 83.42, 60.413, 46.458, -50.505]
  Call Extruder(55.53296)
  MoveL 893 to (-40.24, 47.56, 31.63) mm, rotated rx 180 ry 0 rz 180 deg; joints [-39.027, -20.888, 83.429, 60.365, 46.423, -50.468]
  MoveL 894 to (-40.24, 47.56, 31.63) mm, rotated rx 180 ry 0 rz 180 deg; joints [-39.027, -20.888, 83.429, 60.365, 46.423, -50.468]
  Call Extruder(55.65864)
  MoveL 895 to (-40.2, 47.33, 31.63) mm, rotated rx 180 ry 0 rz 180 deg; joints [-38.982, -20.902, 83.437, 60.321, 46.391, -50.434]
  MoveL 896 to (-40.2, 47.33, 31.63) mm, rotated rx 180 ry 0 rz 180 deg; joints [-38.982, -20.902, 83.437, 60.321, 46.391, -50.434]
  Call Extruder(55.77259)
  MoveL 897 to (-40.15, 47.12, 31.63) mm, rotated rx -180 ry 0 rz 180 deg; joints [-38.941, -20.914, 83.444, 60.281, 46.362, -50.403]
  MoveL 898 to (-40.15, 47.12, 31.63) mm, rotated rx -180 ry 0 rz 180 deg; joints [-38.941, -20.914, 83.444, 60.281, 46.362, -50.403]
  Call Extruder(55.88700)
  MoveL 899 to (-40.11, 46.92, 31.63) mm, rotated rx 180 ry 0 rz 180 deg; joints [-38.9, -20.926, 83.451, 60.241, 46.333, -50.373]
  MoveL 900 to (-40.11, 46.92, 31.63) mm, rotated rx 180 ry 0 rz 180 deg; joints [-38.9, -20.926, 83.451, 60.241, 46.333, -50.373]
  Call Extruder(56.00186)
  MoveL 901 to (-40.06, 46.72, 31.63) mm, rotated rx 180 ry 0 rz 180 deg; joints [-38.859, -20.938, 83.458, 60.201, 46.304, -50.342]
  MoveL 902 to (-40.06, 46.72, 31.63) mm, rotated rx 180 ry 0 rz 180 deg; joints [-38.859, -20.938, 83.458, 60.201, 46.304, -50.342]
  Call Extruder(56.11717)
  MoveL 903 to (-40.02, 46.51, 31.63) mm, rotated rx 180 ry 0 rz 180 deg; joints [-38.819, -20.949, 83.465, 60.161, 46.275, -50.311]
  MoveL 904 to (-40.02, 46.51, 31.63) mm, rotated rx 180 ry 0 rz 180 deg; joints [-38.819, -20.949, 83.465, 60.161, 46.275, -50.311]
  Call Extruder(56.24656)
  MoveL 905 to (-39.95, 46.29, 31.63) mm, rotated rx 180 ry 0 rz 180 deg; joints [-38.771, -20.961, 83.472, 60.115, 46.241, -50.277]
  MoveL 906 to (-39.95, 46.29, 31.63) mm, rotated rx 180 ry 0 rz 180 deg; joints [-38.771, -20.961, 83.472, 60.115, 46.241, -50.277]
  Call Extruder(56.37650)
  MoveL 907 to (-39.88, 46.06, 31.63) mm, rotated rx 180 ry 0 rz 180 deg; joints [-38.724, -20.972, 83.478, 60.069, 46.207, -50.242]
  MoveL 908 to (-39.88, 46.06, 31.63) mm, rotated rx 180 ry 0 rz 180 deg; joints [-38.724, -20.972, 83.478, 60.069, 46.207, -50.242]
  Call Extruder(56.50702)
  MoveL 909 to (-39.81, 45.84, 31.63) mm, rotated rx 180 ry 0 rz 180 deg; joints [-38.677, -20.983, 83.485, 60.023, 46.173, -50.208]
  MoveL 910 to (-39.81, 45.84, 31.63) mm, rotated rx 180 ry 0 rz 180 deg; joints [-38.677, -20.983, 83.485, 60.023, 46.173, -50.208]
  Call Extruder(56.63809)
  MoveL 911 to (-39.75, 45.62, 31.63) mm, rotated rx 180 ry 0 rz 180 deg; joints [-38.629, -20.994, 83.491, 59.978, 46.138, -50.173]
  MoveL 912 to (-39.75, 45.62, 31.63) mm, rotated rx 180 ry 0 rz 180 deg; joints [-38.629, -20.994, 83.491, 59.978, 46.138, -50.173]
  Call Extruder(56.75974)
  MoveL 913 to (-39.68, 45.41, 31.63) mm, rotated rx 180 ry 0 rz 180 deg; joints [-38.585, -21.004, 83.497, 59.935, 46.106, -50.141]
  MoveL 914 to (-39.68, 45.41, 31.63) mm, rotated rx 180 ry 0 rz 180 deg; joints [-38.585, -21.004, 83.497, 59.935, 46.106, -50.141]
  Call Extruder(56.87186)
  MoveL 915 to (-39.62, 45.22, 31.63) mm, rotated rx 180 ry 0 rz -180 deg; joints [-38.544, -21.013, 83.502, 59.896, 46.077, -50.112]
  MoveL 916 to (-39.62, 45.22, 31.63) mm, rotated rx 180 ry 0 rz -180 deg; joints [-38.544, -21.013, 83.502, 59.896, 46.077, -50.112]
  Call Extruder(56.98443)
  MoveL 917 to (-39.56, 45.03, 31.63) mm, rotated rx 180 ry 0 rz 180 deg; joints [-38.504, -21.021, 83.507, 59.857, 46.048, -50.082]
  MoveL 918 to (-39.56, 45.03, 31.63) mm, rotated rx 180 ry 0 rz 180 deg; joints [-38.504, -21.021, 83.507, 59.857, 46.048, -50.082]
  Call Extruder(57.09744)
  MoveL 919 to (-39.5, 44.85, 31.63) mm, rotated rx -180 ry 0 rz 180 deg; joints [-38.463, -21.03, 83.513, 59.817, 46.019, -50.053]
  MoveL 920 to (-39.5, 44.85, 31.63) mm, rotated rx -180 ry 0 rz 180 deg; joints [-38.463, -21.03, 83.513, 59.817, 46.019, -50.053]
  Call Extruder(57.21090)
  MoveL 921 to (-39.44, 44.66, 31.63) mm, rotated rx 180 ry 0 rz -180 deg; joints [-38.422, -21.039, 83.518, 59.778, 45.989, -50.023]
  MoveL 922 to (-39.44, 44.66, 31.63) mm, rotated rx 180 ry 0 rz -180 deg; joints [-38.422, -21.039, 83.518, 59.778, 45.989, -50.023]
  Call Extruder(57.35854)
  MoveL 923 to (-39.35, 44.42, 31.63) mm, rotated rx 180 ry 0 rz 180 deg; joints [-38.369, -21.049, 83.523, 59.727, 45.95, -49.985]
  MoveL 924 to (-39.35, 44.42, 31.63) mm, rotated rx 180 ry 0 rz 180 deg; joints [-38.369, -21.049, 83.523, 59.727, 45.95, -49.985]
  Call Extruder(57.54088)
  MoveL 925 to (-39.23, 44.13, 31.63) mm, rotated rx -180 ry 0 rz 180 deg; joints [-38.302, -21.06, 83.53, 59.663, 45.901, -49.938]
  MoveL 926 to (-39.23, 44.13, 31.63) mm, rotated rx -180 ry 0 rz 180 deg; joints [-38.302, -21.06, 83.53, 59.663, 45.901, -49.938]
  Call Extruder(57.72398)
  MoveL 927 to (-39.11, 43.83, 31.63) mm, rotated rx 180 ry 0 rz 180 deg; joints [-38.236, -21.071, 83.536, 59.6, 45.853, -49.891]
  MoveL 928 to (-39.11, 43.83, 31.63) mm, rotated rx 180 ry 0 rz 180 deg; joints [-38.236, -21.071, 83.536, 59.6, 45.853, -49.891]
  Call Extruder(57.88166)
  MoveL 929 to (-39, 43.58, 31.63) mm, rotated rx -180 ry 0 rz 180 deg; joints [-38.178, -21.08, 83.542, 59.545, 45.811, -49.85]
  MoveL 930 to (-39, 43.58, 31.63) mm, rotated rx -180 ry 0 rz 180 deg; joints [-38.178, -21.08, 83.542, 59.545, 45.811, -49.85]
  Call Extruder(58.03994)
  MoveL 931 to (-38.89, 43.34, 31.63) mm, rotated rx 180 ry 0 rz 180 deg; joints [-38.121, -21.089, 83.547, 59.49, 45.769, -49.81]
  MoveL 932 to (-38.89, 43.34, 31.63) mm, rotated rx 180 ry 0 rz 180 deg; joints [-38.121, -21.089, 83.547, 59.49, 45.769, -49.81]
  Call Extruder(58.22197)
  MoveL 933 to (-38.75, 43.06, 31.63) mm, rotated rx -180 ry 0 rz 180 deg; joints [-38.054, -21.096, 83.551, 59.427, 45.719, -49.764]
  MoveL 934 to (-38.75, 43.06, 31.63) mm, rotated rx -180 ry 0 rz 180 deg; joints [-38.054, -21.096, 83.551, 59.427, 45.719, -49.764]
  Call Extruder(58.42852)
  MoveL 935 to (-38.57, 42.75, 31.63) mm, rotated rx 180 ry 0 rz 180 deg; joints [-37.977, -21.102, 83.555, 59.356, 45.662, -49.713]
  MoveL 936 to (-38.57, 42.75, 31.63) mm, rotated rx 180 ry 0 rz 180 deg; joints [-37.977, -21.102, 83.555, 59.356, 45.662, -49.713]
  Call Extruder(58.63586)
  MoveL 937 to (-38.4, 42.45, 31.63) mm, rotated rx 180 ry 0 rz 180 deg; joints [-37.901, -21.109, 83.559, 59.285, 45.605, -49.661]
  MoveL 938 to (-38.4, 42.45, 31.63) mm, rotated rx 180 ry 0 rz 180 deg; joints [-37.901, -21.109, 83.559, 59.285, 45.605, -49.661]
  Call Extruder(58.84397)
  MoveL 939 to (-38.22, 42.15, 31.63) mm, rotated rx 180 ry 0 rz 180 deg; joints [-37.825, -21.115, 83.562, 59.214, 45.548, -49.61]
  MoveL 940 to (-38.22, 42.15, 31.63) mm, rotated rx 180 ry 0 rz 180 deg; joints [-37.825, -21.115, 83.562, 59.214, 45.548, -49.61]
  Call Extruder(58.96168)
  MoveL 941 to (-38.12, 41.98, 31.63) mm, rotated rx 180 ry 0 rz 180 deg; joints [-37.782, -21.118, 83.564, 59.173, 45.516, -49.581]
  MoveL 942 to (-38.12, 41.98, 31.63) mm, rotated rx 180 ry 0 rz 180 deg; joints [-37.782, -21.118, 83.564, 59.173, 45.516, -49.581]
  Call Extruder(59.29452)
  MoveL 943 to (-37.8, 41.52, 31.63) mm, rotated rx 180 ry 0 rz 180 deg; joints [-37.659, -21.12, 83.565, 59.061, 45.423, -49.501]
  MoveL 944 to (-37.8, 41.52, 31.63) mm, rotated rx 180 ry 0 rz 180 deg; joints [-37.659, -21.12, 83.565, 59.061, 45.423, -49.501]
  Call Extruder(59.62855)
  MoveL 945 to (-37.47, 41.07, 31.63) mm, rotated rx 180 ry 0 rz 180 deg; joints [-37.537, -21.122, 83.566, 58.948, 45.331, -49.422]
  MoveL 946 to (-37.47, 41.07, 31.63) mm, rotated rx 180 ry 0 rz 180 deg; joints [-37.537, -21.122, 83.566, 58.948, 45.331, -49.422]
  Call Extruder(59.79614)
  MoveL 947 to (-37.3, 40.85, 31.63) mm, rotated rx 180 ry 0 rz 180 deg; joints [-37.475, -21.123, 83.567, 58.892, 45.284, -49.382]
  Call Extruder(60.62546)
  MoveL 948 to (-36.39, 39.81, 31.63) mm, rotated rx 180 ry 0 rz 180 deg; joints [-37.173, -21.111, 83.56, 58.618, 45.053, -49.192]
  Call Extruder(61.25652)
  MoveL 949 to (-35.61, 39.11, 31.63) mm, rotated rx 180 ry 0 rz 180 deg; joints [-36.947, -21.084, 83.544, 58.418, 44.876, -49.057]
  MoveL 950 to (-35.61, 39.11, 31.63) mm, rotated rx 180 ry 0 rz 180 deg; joints [-36.947, -21.084, 83.544, 58.418, 44.876, -49.057]
  Call Extruder(61.45410)
  MoveL 951 to (-35.35, 38.9, 31.63) mm, rotated rx 180 ry 0 rz -180 deg; joints [-36.876, -21.075, 83.539, 58.355, 44.821, -49.015]
  Call Extruder(61.78811)
  MoveL 952 to (-34.9, 38.57, 31.63) mm, rotated rx -180 ry 0 rz -180 deg; joints [-36.759, -21.054, 83.527, 58.254, 44.728, -48.948]
  MoveL 953 to (-34.9, 38.57, 31.63) mm, rotated rx -180 ry 0 rz -180 deg; joints [-36.759, -21.054, 83.527, 58.254, 44.728, -48.948]
  Call Extruder(62.12095)
  MoveL 954 to (-34.45, 38.24, 31.63) mm, rotated rx -180 ry 0 rz -180 deg; joints [-36.642, -21.033, 83.514, 58.152, 44.635, -48.881]
  MoveL 955 to (-34.45, 38.24, 31.63) mm, rotated rx -180 ry 0 rz -180 deg; joints [-36.642, -21.033, 83.514, 58.152, 44.635, -48.881]
  Call Extruder(62.30019)
  MoveL 956 to (-34.21, 38.07, 31.63) mm, rotated rx 180 ry 0 rz -180 deg; joints [-36.579, -21.022, 83.507, 58.098, 44.585, -48.845]
  MoveL 957 to (-34.21, 38.07, 31.63) mm, rotated rx 180 ry 0 rz -180 deg; joints [-36.579, -21.022, 83.507, 58.098, 44.585, -48.845]
  Call Extruder(62.50830)
  MoveL 958 to (-33.9, 37.89, 31.63) mm, rotated rx -180 ry 0 rz 180 deg; joints [-36.509, -21.004, 83.497, 58.038, 44.528, -48.806]
  MoveL 959 to (-33.9, 37.89, 31.63) mm, rotated rx -180 ry 0 rz 180 deg; joints [-36.509, -21.004, 83.497, 58.038, 44.528, -48.806]
  Call Extruder(62.71564)
  MoveL 960 to (-33.6, 37.71, 31.63) mm, rotated rx 180 ry 0 rz 180 deg; joints [-36.439, -20.986, 83.487, 57.978, 44.472, -48.768]
  MoveL 961 to (-33.6, 37.71, 31.63) mm, rotated rx 180 ry 0 rz 180 deg; joints [-36.439, -20.986, 83.487, 57.978, 44.472, -48.768]
  Call Extruder(62.92219)
  MoveL 962 to (-33.29, 37.54, 31.63) mm, rotated rx 180 ry 0 rz 180 deg; joints [-36.368, -20.968, 83.476, 57.918, 44.415, -48.73]
  MoveL 963 to (-33.29, 37.54, 31.63) mm, rotated rx 180 ry 0 rz 180 deg; joints [-36.368, -20.968, 83.476, 57.918, 44.415, -48.73]
  Call Extruder(63.12796)
  MoveL 964 to (-32.99, 37.36, 31.63) mm, rotated rx 180 ry 0 rz -180 deg; joints [-36.298, -20.95, 83.465, 57.858, 44.358, -48.691]
  MoveL 965 to (-32.99, 37.36, 31.63) mm, rotated rx 180 ry 0 rz -180 deg; joints [-36.298, -20.95, 83.465, 57.858, 44.358, -48.691]
  Call Extruder(63.28626)
  MoveL 966 to (-32.74, 37.26, 31.63) mm, rotated rx 180 ry 0 rz 180 deg; joints [-36.247, -20.933, 83.455, 57.816, 44.316, -48.666]
  MoveL 967 to (-32.74, 37.26, 31.63) mm, rotated rx 180 ry 0 rz 180 deg; joints [-36.247, -20.933, 83.455, 57.816, 44.316, -48.666]
  Call Extruder(63.44397)
  MoveL 968 to (-32.49, 37.15, 31.63) mm, rotated rx -180 ry 0 rz 180 deg; joints [-36.196, -20.915, 83.445, 57.774, 44.274, -48.64]
  MoveL 969 to (-32.49, 37.15, 31.63) mm, rotated rx -180 ry 0 rz 180 deg; joints [-36.196, -20.915, 83.445, 57.774, 44.274, -48.64]
  Call Extruder(63.61405)
  MoveL 970 to (-32.22, 37.04, 31.63) mm, rotated rx 180 ry 0 rz 180 deg; joints [-36.141, -20.896, 83.433, 57.729, 44.228, -48.612]
  MoveL 971 to (-32.22, 37.04, 31.63) mm, rotated rx 180 ry 0 rz 180 deg; joints [-36.141, -20.896, 83.433, 57.729, 44.228, -48.612]
  Call Extruder(63.79638)
  MoveL 972 to (-31.93, 36.91, 31.63) mm, rotated rx 180 ry 0 rz 180 deg; joints [-36.082, -20.875, 83.421, 57.681, 44.18, -48.582]
  MoveL 973 to (-31.93, 36.91, 31.63) mm, rotated rx 180 ry 0 rz 180 deg; joints [-36.082, -20.875, 83.421, 57.681, 44.18, -48.582]
  Call Extruder(63.97796)
  MoveL 974 to (-31.64, 36.79, 31.63) mm, rotated rx -180 ry 0 rz 180 deg; joints [-36.023, -20.854, 83.409, 57.632, 44.131, -48.553]
  MoveL 975 to (-31.64, 36.79, 31.63) mm, rotated rx -180 ry 0 rz 180 deg; joints [-36.023, -20.854, 83.409, 57.632, 44.131, -48.553]
  Call Extruder(64.09142)
  MoveL 976 to (-31.45, 36.73, 31.63) mm, rotated rx 180 ry 0 rz 180 deg; joints [-35.989, -20.839, 83.4, 57.604, 44.102, -48.536]
  MoveL 977 to (-31.45, 36.73, 31.63) mm, rotated rx 180 ry 0 rz 180 deg; joints [-35.989, -20.839, 83.4, 57.604, 44.102, -48.536]
  Call Extruder(64.20443)
  MoveL 978 to (-31.26, 36.67, 31.63) mm, rotated rx 180 ry 0 rz 180 deg; joints [-35.954, -20.824, 83.391, 57.576, 44.072, -48.52]
  MoveL 979 to (-31.26, 36.67, 31.63) mm, rotated rx 180 ry 0 rz 180 deg; joints [-35.954, -20.824, 83.391, 57.576, 44.072, -48.52]
  Call Extruder(64.31700)
  MoveL 980 to (-31.07, 36.61, 31.63) mm, rotated rx 180 ry 0 rz 180 deg; joints [-35.919, -20.81, 83.382, 57.548, 44.043, -48.503]
  MoveL 981 to (-31.07, 36.61, 31.63) mm, rotated rx 180 ry 0 rz 180 deg; joints [-35.919, -20.81, 83.382, 57.548, 44.043, -48.503]
  Call Extruder(64.42913)
  MoveL 982 to (-30.88, 36.55, 31.63) mm, rotated rx 180 ry 0 rz 180 deg; joints [-35.884, -20.795, 83.373, 57.52, 44.013, -48.487]
  MoveL 983 to (-30.88, 36.55, 31.63) mm, rotated rx 180 ry 0 rz 180 deg; joints [-35.884, -20.795, 83.373, 57.52, 44.013, -48.487]
  Call Extruder(64.54081)
  MoveL 984 to (-30.69, 36.49, 31.63) mm, rotated rx -180 ry 0 rz 180 deg; joints [-35.849, -20.78, 83.365, 57.493, 43.984, -48.47]
  MoveL 985 to (-30.69, 36.49, 31.63) mm, rotated rx -180 ry 0 rz 180 deg; joints [-35.849, -20.78, 83.365, 57.493, 43.984, -48.47]
  Call Extruder(64.67188)
  MoveL 986 to (-30.47, 36.42, 31.63) mm, rotated rx 180 ry 0 rz 180 deg; joints [-35.809, -20.762, 83.354, 57.46, 43.95, -48.451]
  MoveL 987 to (-30.47, 36.42, 31.63) mm, rotated rx 180 ry 0 rz 180 deg; joints [-35.809, -20.762, 83.354, 57.46, 43.95, -48.451]
  Call Extruder(64.80239)
  MoveL 988 to (-30.25, 36.35, 31.63) mm, rotated rx -180 ry 0 rz 180 deg; joints [-35.768, -20.743, 83.343, 57.428, 43.916, -48.433]
  MoveL 989 to (-30.25, 36.35, 31.63) mm, rotated rx -180 ry 0 rz 180 deg; joints [-35.768, -20.743, 83.343, 57.428, 43.916, -48.433]
  Call Extruder(64.93233)
  MoveL 990 to (-30.02, 36.28, 31.63) mm, rotated rx 180 ry 0 rz -180 deg; joints [-35.728, -20.725, 83.333, 57.396, 43.882, -48.414]
  MoveL 991 to (-30.02, 36.28, 31.63) mm, rotated rx 180 ry 0 rz -180 deg; joints [-35.728, -20.725, 83.333, 57.396, 43.882, -48.414]
  Call Extruder(65.06171)
  MoveL 992 to (-29.8, 36.22, 31.63) mm, rotated rx 180 ry 0 rz 180 deg; joints [-35.688, -20.707, 83.322, 57.364, 43.848, -48.395]
  MoveL 993 to (-29.8, 36.22, 31.63) mm, rotated rx 180 ry 0 rz 180 deg; joints [-35.688, -20.707, 83.322, 57.364, 43.848, -48.395]
  Call Extruder(65.18367)
  MoveL 994 to (-29.59, 36.16, 31.63) mm, rotated rx 180 ry 0 rz -180 deg; joints [-35.651, -20.689, 83.311, 57.335, 43.816, -48.378]
  MoveL 995 to (-29.59, 36.16, 31.63) mm, rotated rx 180 ry 0 rz -180 deg; joints [-35.651, -20.689, 83.311, 57.335, 43.816, -48.378]
  Call Extruder(65.29852)
  MoveL 996 to (-29.38, 36.12, 31.63) mm, rotated rx -180 ry 0 rz 180 deg; joints [-35.617, -20.671, 83.3, 57.309, 43.787, -48.364]
  MoveL 997 to (-29.38, 36.12, 31.63) mm, rotated rx -180 ry 0 rz 180 deg; joints [-35.617, -20.671, 83.3, 57.309, 43.787, -48.364]
  Call Extruder(65.41291)
  MoveL 998 to (-29.18, 36.07, 31.63) mm, rotated rx 180 ry 0 rz 180 deg; joints [-35.584, -20.654, 83.29, 57.283, 43.758, -48.349]
  MoveL 999 to (-29.18, 36.07, 31.63) mm, rotated rx 180 ry 0 rz 180 deg; joints [-35.584, -20.654, 83.29, 57.283, 43.758, -48.349]
  Call Extruder(65.52685)
  MoveL 1000 to (-28.97, 36.03, 31.63) mm, rotated rx 180 ry 0 rz 180 deg; joints [-35.55, -20.636, 83.279, 57.257, 43.729, -48.335]
  MoveL 1001 to (-28.97, 36.03, 31.63) mm, rotated rx 180 ry 0 rz 180 deg; joints [-35.55, -20.636, 83.279, 57.257, 43.729, -48.335]
  Call Extruder(65.64034)
  MoveL 1002 to (-28.77, 35.98, 31.63) mm, rotated rx 180 ry 0 rz 180 deg; joints [-35.517, -20.618, 83.268, 57.231, 43.7, -48.32]
  MoveL 1003 to (-28.77, 35.98, 31.63) mm, rotated rx 180 ry 0 rz 180 deg; joints [-35.517, -20.618, 83.268, 57.231, 43.7, -48.32]
  Call Extruder(65.77762)
  MoveL 1004 to (-28.52, 35.93, 31.63) mm, rotated rx -180 ry 0 rz 180 deg; joints [-35.477, -20.596, 83.255, 57.201, 43.665, -48.303]
  MoveL 1005 to (-28.52, 35.93, 31.63) mm, rotated rx -180 ry 0 rz 180 deg; joints [-35.477, -20.596, 83.255, 57.201, 43.665, -48.303]
  Call Extruder(65.91430)
  MoveL 1006 to (-28.27, 35.88, 31.63) mm, rotated rx -180 ry 0 rz 180 deg; joints [-35.437, -20.573, 83.242, 57.17, 43.631, -48.286]
  MoveL 1007 to (-28.27, 35.88, 31.63) mm, rotated rx -180 ry 0 rz 180 deg; joints [-35.437, -20.573, 83.242, 57.17, 43.631, -48.286]
  Call Extruder(66.05036)
  MoveL 1008 to (-28.02, 35.83, 31.63) mm, rotated rx 180 ry 0 rz -180 deg; joints [-35.397, -20.551, 83.229, 57.139, 43.596, -48.269]
  MoveL 1009 to (-28.02, 35.83, 31.63) mm, rotated rx 180 ry 0 rz -180 deg; joints [-35.397, -20.551, 83.229, 57.139, 43.596, -48.269]
  Call Extruder(66.18581)
  MoveL 1010 to (-27.77, 35.78, 31.63) mm, rotated rx 180 ry 0 rz 180 deg; joints [-35.357, -20.529, 83.215, 57.109, 43.562, -48.252]
  MoveL 1011 to (-27.77, 35.78, 31.63) mm, rotated rx 180 ry 0 rz 180 deg; joints [-35.357, -20.529, 83.215, 57.109, 43.562, -48.252]
  Call Extruder(66.32065)
  MoveL 1012 to (-27.52, 35.73, 31.63) mm, rotated rx 180 ry 0 rz 180 deg; joints [-35.317, -20.507, 83.202, 57.078, 43.527, -48.235]
  MoveL 1013 to (-27.52, 35.73, 31.63) mm, rotated rx 180 ry 0 rz 180 deg; joints [-35.317, -20.507, 83.202, 57.078, 43.527, -48.235]
  Call Extruder(66.45488)
  MoveL 1014 to (-27.27, 35.68, 31.63) mm, rotated rx 180 ry 0 rz 180 deg; joints [-35.277, -20.484, 83.189, 57.048, 43.492, -48.218]
  MoveL 1015 to (-27.27, 35.68, 31.63) mm, rotated rx 180 ry 0 rz 180 deg; joints [-35.277, -20.484, 83.189, 57.048, 43.492, -48.218]
  Call Extruder(66.58851)
  MoveL 1016 to (-27.03, 35.64, 31.63) mm, rotated rx -180 ry 0 rz 180 deg; joints [-35.238, -20.462, 83.175, 57.017, 43.458, -48.201]
  MoveL 1017 to (-27.03, 35.64, 31.63) mm, rotated rx -180 ry 0 rz 180 deg; joints [-35.238, -20.462, 83.175, 57.017, 43.458, -48.201]
  Call Extruder(66.75060)
  MoveL 1018 to (-26.72, 35.59, 31.63) mm, rotated rx -180 ry 0 rz 180 deg; joints [-35.191, -20.434, 83.158, 56.982, 43.417, -48.182]
  MoveL 1019 to (-26.72, 35.59, 31.63) mm, rotated rx -180 ry 0 rz 180 deg; joints [-35.191, -20.434, 83.158, 56.982, 43.417, -48.182]
  Call Extruder(66.91198)
  MoveL 1020 to (-26.41, 35.54, 31.63) mm, rotated rx 180 ry 0 rz 180 deg; joints [-35.145, -20.405, 83.141, 56.947, 43.376, -48.164]
  MoveL 1021 to (-26.41, 35.54, 31.63) mm, rotated rx 180 ry 0 rz 180 deg; joints [-35.145, -20.405, 83.141, 56.947, 43.376, -48.164]
  Call Extruder(67.07262)
  MoveL 1022 to (-26.11, 35.49, 31.63) mm, rotated rx 180 ry 0 rz 180 deg; joints [-35.098, -20.377, 83.124, 56.912, 43.336, -48.145]
  MoveL 1023 to (-26.11, 35.49, 31.63) mm, rotated rx 180 ry 0 rz 180 deg; joints [-35.098, -20.377, 83.124, 56.912, 43.336, -48.145]
  Call Extruder(67.23253)
  MoveL 1024 to (-25.8, 35.44, 31.63) mm, rotated rx 180 ry 0 rz 180 deg; joints [-35.052, -20.348, 83.107, 56.877, 43.295, -48.126]
  MoveL 1025 to (-25.8, 35.44, 31.63) mm, rotated rx 180 ry 0 rz 180 deg; joints [-35.052, -20.348, 83.107, 56.877, 43.295, -48.126]
  Call Extruder(67.39172)
  MoveL 1026 to (-25.5, 35.39, 31.63) mm, rotated rx 180 ry 0 rz 180 deg; joints [-35.006, -20.32, 83.09, 56.842, 43.255, -48.107]
  MoveL 1027 to (-25.5, 35.39, 31.63) mm, rotated rx 180 ry 0 rz 180 deg; joints [-35.006, -20.32, 83.09, 56.842, 43.255, -48.107]
  Call Extruder(67.55018)
  MoveL 1028 to (-25.19, 35.34, 31.63) mm, rotated rx 180 ry 0 rz 180 deg; joints [-34.96, -20.291, 83.073, 56.808, 43.214, -48.088]
  MoveL 1029 to (-25.19, 35.34, 31.63) mm, rotated rx 180 ry 0 rz 180 deg; joints [-34.96, -20.291, 83.073, 56.808, 43.214, -48.088]
  Call Extruder(67.74906)
  MoveL 1030 to (-24.8, 35.3, 31.63) mm, rotated rx 180 ry 0 rz 180 deg; joints [-34.904, -20.254, 83.05, 56.767, 43.165, -48.067]
  MoveL 1031 to (-24.8, 35.3, 31.63) mm, rotated rx 180 ry 0 rz 180 deg; joints [-34.904, -20.254, 83.05, 56.767, 43.165, -48.067]
  Call Extruder(67.94707)
  MoveL 1032 to (-24.42, 35.25, 31.63) mm, rotated rx 180 ry 0 rz 180 deg; joints [-34.849, -20.217, 83.028, 56.726, 43.115, -48.045]
  MoveL 1033 to (-24.42, 35.25, 31.63) mm, rotated rx 180 ry 0 rz 180 deg; joints [-34.849, -20.217, 83.028, 56.726, 43.115, -48.045]
  Call Extruder(68.14421)
  MoveL 1034 to (-24.03, 35.21, 31.63) mm, rotated rx 180 ry 0 rz 180 deg; joints [-34.794, -20.179, 83.005, 56.685, 43.066, -48.024]
  MoveL 1035 to (-24.03, 35.21, 31.63) mm, rotated rx 180 ry 0 rz 180 deg; joints [-34.794, -20.179, 83.005, 56.685, 43.066, -48.024]
  Call Extruder(68.34048)
  MoveL 1036 to (-23.64, 35.16, 31.63) mm, rotated rx -180 ry 0 rz 180 deg; joints [-34.738, -20.142, 82.982, 56.644, 43.017, -48.002]
  MoveL 1037 to (-23.64, 35.16, 31.63) mm, rotated rx -180 ry 0 rz 180 deg; joints [-34.738, -20.142, 82.982, 56.644, 43.017, -48.002]
  Call Extruder(68.58617)
  MoveL 1038 to (-23.15, 35.11, 31.63) mm, rotated rx 180 ry 0 rz 180 deg; joints [-34.671, -20.094, 82.953, 56.594, 42.956, -47.977]
  MoveL 1039 to (-23.15, 35.11, 31.63) mm, rotated rx 180 ry 0 rz 180 deg; joints [-34.671, -20.094, 82.953, 56.594, 42.956, -47.977]
  Call Extruder(68.88090)
  MoveL 1040 to (-22.56, 35.07, 31.63) mm, rotated rx -180 ry 0 rz -180 deg; joints [-34.592, -20.035, 82.917, 56.537, 42.885, -47.948]
  MoveL 1041 to (-22.56, 35.07, 31.63) mm, rotated rx -180 ry 0 rz -180 deg; joints [-34.592, -20.035, 82.917, 56.537, 42.885, -47.948]
  Call Extruder(69.17429)
  MoveL 1042 to (-21.97, 35.02, 31.63) mm, rotated rx 180 ry 0 rz 180 deg; joints [-34.512, -19.976, 82.881, 56.48, 42.813, -47.919]
  MoveL 1043 to (-21.97, 35.02, 31.63) mm, rotated rx 180 ry 0 rz 180 deg; joints [-34.512, -19.976, 82.881, 56.48, 42.813, -47.919]
  Call Extruder(69.60762)
  MoveL 1044 to (-21.1, 34.97, 31.63) mm, rotated rx 180 ry 0 rz 180 deg; joints [-34.399, -19.887, 82.827, 56.399, 42.71, -47.88]
  MoveL 1045 to (-21.1, 34.97, 31.63) mm, rotated rx 180 ry 0 rz 180 deg; joints [-34.399, -19.887, 82.827, 56.399, 42.71, -47.88]
  Call Extruder(70.17978)
  MoveL 1046 to (-19.94, 34.93, 31.63) mm, rotated rx 180 ry 0 rz 180 deg; joints [-34.253, -19.767, 82.753, 56.296, 42.576, -47.83]
  MoveL 1047 to (-19.94, 34.93, 31.63) mm, rotated rx 180 ry 0 rz 180 deg; joints [-34.253, -19.767, 82.753, 56.296, 42.576, -47.83]
  Call Extruder(70.60761)
  MoveL 1048 to (-19.06, 34.91, 31.63) mm, rotated rx -180 ry 0 rz 180 deg; joints [-34.146, -19.675, 82.697, 56.222, 42.477, -47.795]
  Call Extruder(187.25630)
  MoveL 1049 to (219.06, 34.91, 31.63) mm, rotated rx 180 ry 0 rz 180 deg; joints [-18.248, 13.245, 51.824, 38.032, 30.548, -33.965]
  MoveL 1050 to (219.06, 34.91, 31.63) mm, rotated rx 180 ry 0 rz 180 deg; joints [-18.248, 13.245, 51.824, 38.032, 30.548, -33.965]
  Call Extruder(187.97187)
  MoveL 1051 to (220.52, 34.95, 31.63) mm, rotated rx -180 ry 0 rz 180 deg; joints [-18.199, 13.52, 51.478, 37.879, 30.576, -33.811]
  MoveL 1052 to (220.52, 34.95, 31.63) mm, rotated rx -180 ry 0 rz 180 deg; joints [-18.199, 13.52, 51.478, 37.879, 30.576, -33.811]
  Call Extruder(188.54661)
  MoveL 1053 to (221.68, 35, 31.63) mm, rotated rx 180 ry 0 rz 180 deg; joints [-18.162, 13.742, 51.198, 37.757, 30.601, -33.689]
  MoveL 1054 to (221.68, 35, 31.63) mm, rotated rx 180 ry 0 rz 180 deg; joints [-18.162, 13.742, 51.198, 37.757, 30.601, -33.689]
  Call Extruder(188.84000)
  MoveL 1055 to (222.27, 35.04, 31.63) mm, rotated rx 180 ry 0 rz 180 deg; joints [-18.146, 13.857, 51.053, 37.7, 30.616, -33.629]
  MoveL 1056 to (222.27, 35.04, 31.63) mm, rotated rx 180 ry 0 rz 180 deg; joints [-18.146, 13.857, 51.053, 37.7, 30.616, -33.629]
  Call Extruder(189.13473)
  MoveL 1057 to (222.86, 35.09, 31.63) mm, rotated rx -180 ry 0 rz 180 deg; joints [-18.13, 13.972, 50.907, 37.641, 30.631, -33.57]
  MoveL 1058 to (222.86, 35.09, 31.63) mm, rotated rx -180 ry 0 rz 180 deg; joints [-18.13, 13.972, 50.907, 37.641, 30.631, -33.57]
  Call Extruder(189.43079)
  MoveL 1059 to (223.45, 35.14, 31.63) mm, rotated rx 180 ry 0 rz 180 deg; joints [-18.113, 14.087, 50.761, 37.583, 30.647, -33.51]
  MoveL 1060 to (223.45, 35.14, 31.63) mm, rotated rx 180 ry 0 rz 180 deg; joints [-18.113, 14.087, 50.761, 37.583, 30.647, -33.51]
  Call Extruder(189.62706)
  MoveL 1061 to (223.84, 35.18, 31.63) mm, rotated rx -180 ry 0 rz 180 deg; joints [-18.104, 14.164, 50.663, 37.547, 30.659, -33.472]
  MoveL 1062 to (223.84, 35.18, 31.63) mm, rotated rx -180 ry 0 rz 180 deg; joints [-18.104, 14.164, 50.663, 37.547, 30.659, -33.472]
  Call Extruder(189.82420)
  MoveL 1063 to (224.22, 35.23, 31.63) mm, rotated rx 180 ry 0 rz 180 deg; joints [-18.095, 14.241, 50.565, 37.51, 30.67, -33.434]
  MoveL 1064 to (224.22, 35.23, 31.63) mm, rotated rx 180 ry 0 rz 180 deg; joints [-18.095, 14.241, 50.565, 37.51, 30.67, -33.434]
  Call Extruder(190.02221)
  MoveL 1065 to (224.61, 35.27, 31.63) mm, rotated rx -180 ry 0 rz 180 deg; joints [-18.087, 14.318, 50.467, 37.474, 30.682, -33.397]
  MoveL 1066 to (224.61, 35.27, 31.63) mm, rotated rx -180 ry 0 rz 180 deg; joints [-18.087, 14.318, 50.467, 37.474, 30.682, -33.397]
  Call Extruder(190.22109)
  MoveL 1067 to (225, 35.32, 31.63) mm, rotated rx -180 ry 0 rz -180 deg; joints [-18.078, 14.395, 50.368, 37.438, 30.694, -33.359]
  MoveL 1068 to (225, 35.32, 31.63) mm, rotated rx -180 ry 0 rz -180 deg; joints [-18.078, 14.395, 50.368, 37.438, 30.694, -33.359]
  Call Extruder(190.40017)
  MoveL 1069 to (225.34, 35.37, 31.63) mm, rotated rx 180 ry 0 rz 180 deg; joints [-18.07, 14.465, 50.279, 37.406, 30.706, -33.325]
  MoveL 1070 to (225.34, 35.37, 31.63) mm, rotated rx 180 ry 0 rz 180 deg; joints [-18.07, 14.465, 50.279, 37.406, 30.706, -33.325]
  Call Extruder(190.55935)
  MoveL 1071 to (225.65, 35.42, 31.63) mm, rotated rx 180 ry 0 rz 180 deg; joints [-18.065, 14.527, 50.2, 37.379, 30.716, -33.297]
  MoveL 1072 to (225.65, 35.42, 31.63) mm, rotated rx 180 ry 0 rz 180 deg; joints [-18.065, 14.527, 50.2, 37.379, 30.716, -33.297]
  Call Extruder(190.71926)
  MoveL 1073 to (225.96, 35.47, 31.63) mm, rotated rx 180 ry 0 rz 180 deg; joints [-18.059, 14.589, 50.12, 37.352, 30.727, -33.268]
  MoveL 1074 to (225.96, 35.47, 31.63) mm, rotated rx 180 ry 0 rz 180 deg; joints [-18.059, 14.589, 50.12, 37.352, 30.727, -33.268]
  Call Extruder(190.87990)
  MoveL 1075 to (226.26, 35.51, 31.63) mm, rotated rx 180 ry 0 rz 180 deg; joints [-18.054, 14.651, 50.041, 37.325, 30.738, -33.24]
  MoveL 1076 to (226.26, 35.51, 31.63) mm, rotated rx 180 ry 0 rz 180 deg; joints [-18.054, 14.651, 50.041, 37.325, 30.738, -33.24]
  Call Extruder(191.04127)
  MoveL 1077 to (226.57, 35.56, 31.63) mm, rotated rx -180 ry 0 rz -180 deg; joints [-18.048, 14.713, 49.961, 37.298, 30.749, -33.211]
  MoveL 1078 to (226.57, 35.56, 31.63) mm, rotated rx -180 ry 0 rz -180 deg; joints [-18.048, 14.713, 49.961, 37.298, 30.749, -33.211]
  Call Extruder(191.20337)
  MoveL 1079 to (226.87, 35.61, 31.63) mm, rotated rx 180 ry 0 rz 180 deg; joints [-18.042, 14.776, 49.881, 37.271, 30.76, -33.182]
  MoveL 1080 to (226.87, 35.61, 31.63) mm, rotated rx 180 ry 0 rz 180 deg; joints [-18.042, 14.776, 49.881, 37.271, 30.76, -33.182]
  Call Extruder(191.35156)
  MoveL 1081 to (227.15, 35.66, 31.63) mm, rotated rx 180 ry 0 rz 180 deg; joints [-18.038, 14.833, 49.808, 37.247, 30.77, -33.156]
  MoveL 1082 to (227.15, 35.66, 31.63) mm, rotated rx 180 ry 0 rz 180 deg; joints [-18.038, 14.833, 49.808, 37.247, 30.77, -33.156]
  Call Extruder(191.48580)
  MoveL 1083 to (227.4, 35.71, 31.63) mm, rotated rx -180 ry 0 rz 180 deg; joints [-18.034, 14.884, 49.741, 37.226, 30.78, -33.134]
  MoveL 1084 to (227.4, 35.71, 31.63) mm, rotated rx -180 ry 0 rz 180 deg; joints [-18.034, 14.884, 49.741, 37.226, 30.78, -33.134]
  Call Extruder(191.62064)
  MoveL 1085 to (227.65, 35.76, 31.63) mm, rotated rx -180 ry 0 rz 180 deg; joints [-18.031, 14.936, 49.675, 37.206, 30.79, -33.112]
  MoveL 1086 to (227.65, 35.76, 31.63) mm, rotated rx -180 ry 0 rz 180 deg; joints [-18.031, 14.936, 49.675, 37.206, 30.79, -33.112]
  Call Extruder(191.75609)
  MoveL 1087 to (227.9, 35.81, 31.63) mm, rotated rx 180 ry 0 rz 180 deg; joints [-18.027, 14.988, 49.608, 37.185, 30.8, -33.089]
  MoveL 1088 to (227.9, 35.81, 31.63) mm, rotated rx 180 ry 0 rz 180 deg; joints [-18.027, 14.988, 49.608, 37.185, 30.8, -33.089]
  Call Extruder(191.89216)
  MoveL 1089 to (228.15, 35.86, 31.63) mm, rotated rx -180 ry 0 rz 180 deg; joints [-18.024, 15.04, 49.541, 37.164, 30.81, -33.067]
  MoveL 1090 to (228.15, 35.86, 31.63) mm, rotated rx -180 ry 0 rz 180 deg; joints [-18.024, 15.04, 49.541, 37.164, 30.81, -33.067]
  Call Extruder(192.02883)
  MoveL 1091 to (228.4, 35.91, 31.63) mm, rotated rx 180 ry 0 rz 180 deg; joints [-18.02, 15.092, 49.474, 37.143, 30.82, -33.044]
  MoveL 1092 to (228.4, 35.91, 31.63) mm, rotated rx 180 ry 0 rz 180 deg; joints [-18.02, 15.092, 49.474, 37.143, 30.82, -33.044]
  Call Extruder(192.16611)
  MoveL 1093 to (228.65, 35.96, 31.63) mm, rotated rx 180 ry 0 rz -180 deg; joints [-18.017, 15.144, 49.407, 37.122, 30.83, -33.021]
  MoveL 1094 to (228.65, 35.96, 31.63) mm, rotated rx 180 ry 0 rz -180 deg; joints [-18.017, 15.144, 49.407, 37.122, 30.83, -33.021]
  Call Extruder(192.29179)
  MoveL 1095 to (228.87, 36, 31.63) mm, rotated rx 180 ry 0 rz 180 deg; joints [-18.014, 15.191, 49.346, 37.103, 30.84, -33.001]
  MoveL 1096 to (228.87, 36, 31.63) mm, rotated rx 180 ry 0 rz 180 deg; joints [-18.014, 15.191, 49.346, 37.103, 30.84, -33.001]
  Call Extruder(192.40573)
  MoveL 1097 to (229.08, 36.05, 31.63) mm, rotated rx 180 ry 0 rz 180 deg; joints [-18.012, 15.234, 49.29, 37.087, 30.848, -32.983]
  MoveL 1098 to (229.08, 36.05, 31.63) mm, rotated rx 180 ry 0 rz 180 deg; joints [-18.012, 15.234, 49.29, 37.087, 30.848, -32.983]
  Call Extruder(192.52012)
  MoveL 1099 to (229.28, 36.09, 31.63) mm, rotated rx 180 ry 0 rz 180 deg; joints [-18.009, 15.277, 49.235, 37.07, 30.857, -32.965]
  MoveL 1100 to (229.28, 36.09, 31.63) mm, rotated rx 180 ry 0 rz 180 deg; joints [-18.009, 15.277, 49.235, 37.07, 30.857, -32.965]
  Call Extruder(192.63497)
  MoveL 1101 to (229.48, 36.14, 31.63) mm, rotated rx 180 ry 0 rz 180 deg; joints [-18.007, 15.32, 49.179, 37.053, 30.866, -32.946]
  MoveL 1102 to (229.48, 36.14, 31.63) mm, rotated rx 180 ry 0 rz 180 deg; joints [-18.007, 15.32, 49.179, 37.053, 30.866, -32.946]
  Call Extruder(192.75028)
  MoveL 1103 to (229.69, 36.18, 31.63) mm, rotated rx 180 ry 0 rz 180 deg; joints [-18.005, 15.363, 49.123, 37.037, 30.875, -32.928]
  MoveL 1104 to (229.69, 36.18, 31.63) mm, rotated rx 180 ry 0 rz 180 deg; joints [-18.005, 15.363, 49.123, 37.037, 30.875, -32.928]
  Call Extruder(192.87966)
  MoveL 1105 to (229.91, 36.25, 31.63) mm, rotated rx 180 ry 0 rz 180 deg; joints [-18.004, 15.412, 49.06, 37.021, 30.886, -32.91]
  MoveL 1106 to (229.91, 36.25, 31.63) mm, rotated rx 180 ry 0 rz 180 deg; joints [-18.004, 15.412, 49.06, 37.021, 30.886, -32.91]
  Call Extruder(193.00961)
  MoveL 1107 to (230.14, 36.32, 31.63) mm, rotated rx 180 ry 0 rz -180 deg; joints [-18.003, 15.46, 48.997, 37.006, 30.897, -32.893]
  MoveL 1108 to (230.14, 36.32, 31.63) mm, rotated rx 180 ry 0 rz -180 deg; joints [-18.003, 15.46, 48.997, 37.006, 30.897, -32.893]
  Call Extruder(193.14012)
  MoveL 1109 to (230.36, 36.39, 31.63) mm, rotated rx 180 ry 0 rz 180 deg; joints [-18.003, 15.509, 48.934, 36.99, 30.909, -32.875]
  MoveL 1110 to (230.36, 36.39, 31.63) mm, rotated rx 180 ry 0 rz 180 deg; joints [-18.003, 15.509, 48.934, 36.99, 30.909, -32.875]
  Call Extruder(193.27120)
  MoveL 1111 to (230.58, 36.45, 31.63) mm, rotated rx 180 ry 0 rz 180 deg; joints [-18.002, 15.558, 48.871, 36.975, 30.92, -32.857]
  MoveL 1112 to (230.58, 36.45, 31.63) mm, rotated rx 180 ry 0 rz 180 deg; joints [-18.002, 15.558, 48.871, 36.975, 30.92, -32.857]
  Call Extruder(193.39284)
  MoveL 1113 to (230.79, 36.52, 31.63) mm, rotated rx 180 ry 0 rz 180 deg; joints [-18.002, 15.603, 48.812, 36.961, 30.931, -32.841]
  MoveL 1114 to (230.79, 36.52, 31.63) mm, rotated rx 180 ry 0 rz 180 deg; joints [-18.002, 15.603, 48.812, 36.961, 30.931, -32.841]
  Call Extruder(193.50496)
  MoveL 1115 to (230.98, 36.58, 31.63) mm, rotated rx -180 ry 0 rz -180 deg; joints [-18.002, 15.644, 48.759, 36.948, 30.941, -32.826]
  MoveL 1116 to (230.98, 36.58, 31.63) mm, rotated rx -180 ry 0 rz -180 deg; joints [-18.002, 15.644, 48.759, 36.948, 30.941, -32.826]
  Call Extruder(193.61753)
  MoveL 1117 to (231.17, 36.64, 31.63) mm, rotated rx 180 ry 0 rz 180 deg; joints [-18.002, 15.685, 48.704, 36.936, 30.951, -32.812]
  MoveL 1118 to (231.17, 36.64, 31.63) mm, rotated rx 180 ry 0 rz 180 deg; joints [-18.002, 15.685, 48.704, 36.936, 30.951, -32.812]
  Call Extruder(193.73054)
  MoveL 1119 to (231.35, 36.7, 31.63) mm, rotated rx 180 ry 0 rz 180 deg; joints [-18.002, 15.727, 48.651, 36.923, 30.961, -32.797]
  MoveL 1120 to (231.35, 36.7, 31.63) mm, rotated rx 180 ry 0 rz 180 deg; joints [-18.002, 15.727, 48.651, 36.923, 30.961, -32.797]
  Call Extruder(193.84399)
  MoveL 1121 to (231.54, 36.76, 31.63) mm, rotated rx 180 ry 0 rz 180 deg; joints [-18.002, 15.768, 48.596, 36.91, 30.971, -32.782]
  MoveL 1122 to (231.54, 36.76, 31.63) mm, rotated rx 180 ry 0 rz 180 deg; joints [-18.002, 15.768, 48.596, 36.91, 30.971, -32.782]
  Call Extruder(193.99163)
  MoveL 1123 to (231.78, 36.85, 31.63) mm, rotated rx 180 ry 0 rz -180 deg; joints [-18.004, 15.822, 48.526, 36.896, 30.985, -32.765]
  MoveL 1124 to (231.78, 36.85, 31.63) mm, rotated rx 180 ry 0 rz -180 deg; joints [-18.004, 15.822, 48.526, 36.896, 30.985, -32.765]
  Call Extruder(194.17397)
  MoveL 1125 to (232.08, 36.98, 31.63) mm, rotated rx -180 ry 0 rz 180 deg; joints [-18.006, 15.888, 48.44, 36.881, 31.002, -32.746]
  MoveL 1126 to (232.08, 36.98, 31.63) mm, rotated rx -180 ry 0 rz 180 deg; joints [-18.006, 15.888, 48.44, 36.881, 31.002, -32.746]
  Call Extruder(194.35707)
  MoveL 1127 to (232.37, 37.1, 31.63) mm, rotated rx 180 ry 0 rz 180 deg; joints [-18.009, 15.955, 48.353, 36.865, 31.02, -32.726]
  MoveL 1128 to (232.37, 37.1, 31.63) mm, rotated rx 180 ry 0 rz 180 deg; joints [-18.009, 15.955, 48.353, 36.865, 31.02, -32.726]
  Call Extruder(194.51476)
  MoveL 1129 to (232.62, 37.2, 31.63) mm, rotated rx -180 ry 0 rz 180 deg; joints [-18.012, 16.012, 48.279, 36.852, 31.036, -32.709]
  MoveL 1130 to (232.62, 37.2, 31.63) mm, rotated rx -180 ry 0 rz 180 deg; joints [-18.012, 16.012, 48.279, 36.852, 31.036, -32.709]
  Call Extruder(194.67306)
  MoveL 1131 to (232.87, 37.31, 31.63) mm, rotated rx 180 ry 0 rz 180 deg; joints [-18.015, 16.069, 48.204, 36.839, 31.051, -32.693]
  MoveL 1132 to (232.87, 37.31, 31.63) mm, rotated rx 180 ry 0 rz 180 deg; joints [-18.015, 16.069, 48.204, 36.839, 31.051, -32.693]
  Call Extruder(194.85509)
  MoveL 1133 to (233.14, 37.45, 31.63) mm, rotated rx 180 ry 0 rz 180 deg; joints [-18.02, 16.134, 48.119, 36.828, 31.071, -32.677]
  MoveL 1134 to (233.14, 37.45, 31.63) mm, rotated rx 180 ry 0 rz 180 deg; joints [-18.02, 16.134, 48.119, 36.828, 31.071, -32.677]
  Call Extruder(195.06165)
  MoveL 1135 to (233.45, 37.63, 31.63) mm, rotated rx 180 ry 0 rz 180 deg; joints [-18.029, 16.206, 48.023, 36.819, 31.093, -32.662]
  MoveL 1136 to (233.45, 37.63, 31.63) mm, rotated rx 180 ry 0 rz 180 deg; joints [-18.029, 16.206, 48.023, 36.819, 31.093, -32.662]
  Call Extruder(195.26898)
  MoveL 1137 to (233.75, 37.8, 31.63) mm, rotated rx -180 ry 0 rz 180 deg; joints [-18.037, 16.279, 47.927, 36.81, 31.116, -32.647]
  MoveL 1138 to (233.75, 37.8, 31.63) mm, rotated rx -180 ry 0 rz 180 deg; joints [-18.037, 16.279, 47.927, 36.81, 31.116, -32.647]
  Call Extruder(195.47710)
  MoveL 1139 to (234.05, 37.98, 31.63) mm, rotated rx -180 ry 0 rz 180 deg; joints [-18.045, 16.352, 47.831, 36.801, 31.139, -32.632]
  MoveL 1140 to (234.05, 37.98, 31.63) mm, rotated rx -180 ry 0 rz 180 deg; joints [-18.045, 16.352, 47.831, 36.801, 31.139, -32.632]
  Call Extruder(195.59482)
  MoveL 1141 to (234.22, 38.08, 31.63) mm, rotated rx -180 ry 0 rz -180 deg; joints [-18.05, 16.394, 47.777, 36.795, 31.152, -32.624]
  MoveL 1142 to (234.22, 38.08, 31.63) mm, rotated rx -180 ry 0 rz -180 deg; joints [-18.05, 16.394, 47.777, 36.795, 31.152, -32.624]
  Call Extruder(195.92764)
  MoveL 1143 to (234.68, 38.41, 31.63) mm, rotated rx -180 ry 0 rz 180 deg; joints [-18.07, 16.507, 47.627, 36.791, 31.191, -32.609]
  MoveL 1144 to (234.68, 38.41, 31.63) mm, rotated rx -180 ry 0 rz 180 deg; joints [-18.07, 16.507, 47.627, 36.791, 31.191, -32.609]
  Call Extruder(196.26165)
  MoveL 1145 to (235.13, 38.73, 31.63) mm, rotated rx -180 ry 0 rz -180 deg; joints [-18.089, 16.621, 47.477, 36.787, 31.231, -32.594]
  MoveL 1146 to (235.13, 38.73, 31.63) mm, rotated rx -180 ry 0 rz -180 deg; joints [-18.089, 16.621, 47.477, 36.787, 31.231, -32.594]
  Call Extruder(196.42923)
  MoveL 1147 to (235.35, 38.9, 31.63) mm, rotated rx -180 ry 0 rz -180 deg; joints [-18.099, 16.678, 47.402, 36.785, 31.251, -32.587]
  Call Extruder(197.25856)
  MoveL 1148 to (236.39, 39.81, 31.63) mm, rotated rx -180 ry 0 rz 180 deg; joints [-18.16, 16.952, 47.039, 36.797, 31.356, -32.569]
  Call Extruder(197.88962)
  MoveL 1149 to (237.09, 40.6, 31.63) mm, rotated rx 180 ry 0 rz 180 deg; joints [-18.22, 17.149, 46.776, 36.83, 31.44, -32.577]
  MoveL 1150 to (237.09, 40.6, 31.63) mm, rotated rx 180 ry 0 rz 180 deg; joints [-18.22, 17.149, 46.776, 36.83, 31.44, -32.577]
  Call Extruder(198.08723)
  MoveL 1151 to (237.3, 40.85, 31.63) mm, rotated rx 180 ry 0 rz 180 deg; joints [-18.24, 17.211, 46.694, 36.841, 31.467, -32.58]
  Call Extruder(198.42124)
  MoveL 1152 to (237.63, 41.3, 31.63) mm, rotated rx 180 ry 0 rz 180 deg; joints [-18.277, 17.31, 46.562, 36.868, 31.513, -32.593]
  MoveL 1153 to (237.63, 41.3, 31.63) mm, rotated rx 180 ry 0 rz 180 deg; joints [-18.277, 17.31, 46.562, 36.868, 31.513, -32.593]
  Call Extruder(198.75406)
  MoveL 1154 to (237.96, 41.75, 31.63) mm, rotated rx 180 ry 0 rz 180 deg; joints [-18.313, 17.409, 46.429, 36.895, 31.56, -32.605]
  MoveL 1155 to (237.96, 41.75, 31.63) mm, rotated rx 180 ry 0 rz 180 deg; joints [-18.313, 17.409, 46.429, 36.895, 31.56, -32.605]
  Call Extruder(198.93329)
  MoveL 1156 to (238.14, 41.99, 31.63) mm, rotated rx 180 ry 0 rz 180 deg; joints [-18.333, 17.463, 46.357, 36.909, 31.585, -32.612]
  MoveL 1157 to (238.14, 41.99, 31.63) mm, rotated rx 180 ry 0 rz 180 deg; joints [-18.333, 17.463, 46.357, 36.909, 31.585, -32.612]
  Call Extruder(199.14141)
  MoveL 1158 to (238.31, 42.3, 31.63) mm, rotated rx 180 ry 0 rz 180 deg; joints [-18.36, 17.521, 46.28, 36.932, 31.615, -32.625]
  MoveL 1159 to (238.31, 42.3, 31.63) mm, rotated rx 180 ry 0 rz 180 deg; joints [-18.36, 17.521, 46.28, 36.932, 31.615, -32.625]
  Call Extruder(199.34875)
  MoveL 1160 to (238.49, 42.6, 31.63) mm, rotated rx 180 ry 0 rz 180 deg; joints [-18.386, 17.579, 46.203, 36.955, 31.645, -32.639]
  MoveL 1161 to (238.49, 42.6, 31.63) mm, rotated rx 180 ry 0 rz 180 deg; joints [-18.386, 17.579, 46.203, 36.955, 31.645, -32.639]
  Call Extruder(199.55531)
  MoveL 1162 to (238.66, 42.91, 31.63) mm, rotated rx 180 ry 0 rz 180 deg; joints [-18.412, 17.637, 46.125, 36.978, 31.675, -32.652]
  MoveL 1163 to (238.66, 42.91, 31.63) mm, rotated rx 180 ry 0 rz 180 deg; joints [-18.412, 17.637, 46.125, 36.978, 31.675, -32.652]
  Call Extruder(199.76109)
  MoveL 1164 to (238.84, 43.21, 31.63) mm, rotated rx 180 ry 0 rz 180 deg; joints [-18.438, 17.695, 46.047, 37.001, 31.705, -32.665]
  MoveL 1165 to (238.84, 43.21, 31.63) mm, rotated rx 180 ry 0 rz 180 deg; joints [-18.438, 17.695, 46.047, 37.001, 31.705, -32.665]
  Call Extruder(199.91939)
  MoveL 1166 to (238.94, 43.46, 31.63) mm, rotated rx 180 ry 0 rz 180 deg; joints [-18.461, 17.735, 45.993, 37.024, 31.728, -32.68]
  MoveL 1167 to (238.94, 43.46, 31.63) mm, rotated rx 180 ry 0 rz 180 deg; joints [-18.461, 17.735, 45.993, 37.024, 31.728, -32.68]
  Call Extruder(200.07710)
  MoveL 1168 to (239.05, 43.71, 31.63) mm, rotated rx -180 ry 0 rz 180 deg; joints [-18.484, 17.775, 45.939, 37.047, 31.751, -32.695]
  MoveL 1169 to (239.05, 43.71, 31.63) mm, rotated rx -180 ry 0 rz 180 deg; joints [-18.484, 17.775, 45.939, 37.047, 31.751, -32.695]
  Call Extruder(200.24718)
  MoveL 1170 to (239.16, 43.98, 31.63) mm, rotated rx -180 ry 0 rz 180 deg; joints [-18.509, 17.818, 45.881, 37.072, 31.776, -32.712]
  MoveL 1171 to (239.16, 43.98, 31.63) mm, rotated rx -180 ry 0 rz 180 deg; joints [-18.509, 17.818, 45.881, 37.072, 31.776, -32.712]
  Call Extruder(200.42950)
  MoveL 1172 to (239.29, 44.27, 31.63) mm, rotated rx -180 ry 0 rz -180 deg; joints [-18.535, 17.864, 45.819, 37.099, 31.804, -32.73]
  MoveL 1173 to (239.29, 44.27, 31.63) mm, rotated rx -180 ry 0 rz -180 deg; joints [-18.535, 17.864, 45.819, 37.099, 31.804, -32.73]
  Call Extruder(200.61107)
  MoveL 1174 to (239.41, 44.56, 31.63) mm, rotated rx -180 ry 0 rz 180 deg; joints [-18.562, 17.91, 45.757, 37.126, 31.831, -32.748]
  MoveL 1175 to (239.41, 44.56, 31.63) mm, rotated rx -180 ry 0 rz 180 deg; joints [-18.562, 17.91, 45.757, 37.126, 31.831, -32.748]
  Call Extruder(200.72453)
  MoveL 1176 to (239.47, 44.75, 31.63) mm, rotated rx 180 ry 0 rz 180 deg; joints [-18.58, 17.937, 45.721, 37.146, 31.848, -32.761]
  MoveL 1177 to (239.47, 44.75, 31.63) mm, rotated rx 180 ry 0 rz 180 deg; joints [-18.58, 17.937, 45.721, 37.146, 31.848, -32.761]
  Call Extruder(200.83755)
  MoveL 1178 to (239.53, 44.94, 31.63) mm, rotated rx -180 ry 0 rz 180 deg; joints [-18.598, 17.963, 45.686, 37.165, 31.865, -32.775]
  MoveL 1179 to (239.53, 44.94, 31.63) mm, rotated rx -180 ry 0 rz 180 deg; joints [-18.598, 17.963, 45.686, 37.165, 31.865, -32.775]
  Call Extruder(200.95013)
  MoveL 1180 to (239.59, 45.13, 31.63) mm, rotated rx -180 ry 0 rz -180 deg; joints [-18.616, 17.99, 45.65, 37.185, 31.882, -32.789]
  MoveL 1181 to (239.59, 45.13, 31.63) mm, rotated rx -180 ry 0 rz -180 deg; joints [-18.616, 17.99, 45.65, 37.185, 31.882, -32.789]
  Call Extruder(201.06226)
  MoveL 1182 to (239.65, 45.32, 31.63) mm, rotated rx 180 ry 0 rz 180 deg; joints [-18.634, 18.016, 45.614, 37.204, 31.899, -32.802]
  MoveL 1183 to (239.65, 45.32, 31.63) mm, rotated rx 180 ry 0 rz 180 deg; joints [-18.634, 18.016, 45.614, 37.204, 31.899, -32.802]
  Call Extruder(201.17395)
  MoveL 1184 to (239.71, 45.5, 31.63) mm, rotated rx 180 ry 0 rz 180 deg; joints [-18.651, 18.042, 45.579, 37.224, 31.916, -32.816]
  MoveL 1185 to (239.71, 45.5, 31.63) mm, rotated rx 180 ry 0 rz 180 deg; joints [-18.651, 18.042, 45.579, 37.224, 31.916, -32.816]
  Call Extruder(201.30502)
  MoveL 1186 to (239.78, 45.73, 31.63) mm, rotated rx -180 ry 0 rz 180 deg; joints [-18.673, 18.073, 45.537, 37.247, 31.936, -32.832]
  MoveL 1187 to (239.78, 45.73, 31.63) mm, rotated rx -180 ry 0 rz 180 deg; joints [-18.673, 18.073, 45.537, 37.247, 31.936, -32.832]
  Call Extruder(201.43553)
  MoveL 1188 to (239.85, 45.95, 31.63) mm, rotated rx 180 ry 0 rz 180 deg; joints [-18.694, 18.103, 45.496, 37.271, 31.956, -32.849]
  MoveL 1189 to (239.85, 45.95, 31.63) mm, rotated rx 180 ry 0 rz 180 deg; joints [-18.694, 18.103, 45.496, 37.271, 31.956, -32.849]
  Call Extruder(201.56547)
  MoveL 1190 to (239.92, 46.18, 31.63) mm, rotated rx -180 ry 0 rz -180 deg; joints [-18.715, 18.134, 45.455, 37.294, 31.976, -32.865]
  MoveL 1191 to (239.92, 46.18, 31.63) mm, rotated rx -180 ry 0 rz -180 deg; joints [-18.715, 18.134, 45.455, 37.294, 31.976, -32.865]
  Call Extruder(201.69485)
  MoveL 1192 to (239.98, 46.4, 31.63) mm, rotated rx -180 ry 0 rz 180 deg; joints [-18.737, 18.164, 45.414, 37.317, 31.996, -32.882]
  MoveL 1193 to (239.98, 46.4, 31.63) mm, rotated rx -180 ry 0 rz 180 deg; joints [-18.737, 18.164, 45.414, 37.317, 31.996, -32.882]
  Call Extruder(201.81681)
  MoveL 1194 to (240.04, 46.61, 31.63) mm, rotated rx 180 ry 0 rz 180 deg; joints [-18.757, 18.192, 45.377, 37.341, 32.015, -32.898]
  MoveL 1195 to (240.04, 46.61, 31.63) mm, rotated rx 180 ry 0 rz 180 deg; joints [-18.757, 18.192, 45.377, 37.341, 32.015, -32.898]
  Call Extruder(201.93163)
  MoveL 1196 to (240.08, 46.82, 31.63) mm, rotated rx 180 ry 0 rz 180 deg; joints [-18.777, 18.216, 45.344, 37.364, 32.033, -32.915]
  MoveL 1197 to (240.08, 46.82, 31.63) mm, rotated rx 180 ry 0 rz 180 deg; joints [-18.777, 18.216, 45.344, 37.364, 32.033, -32.915]
  Call Extruder(202.04601)
  MoveL 1198 to (240.13, 47.02, 31.63) mm, rotated rx 180 ry 0 rz 180 deg; joints [-18.797, 18.24, 45.311, 37.387, 32.051, -32.932]
  MoveL 1199 to (240.13, 47.02, 31.63) mm, rotated rx 180 ry 0 rz 180 deg; joints [-18.797, 18.24, 45.311, 37.387, 32.051, -32.932]
  Call Extruder(202.15993)
  MoveL 1200 to (240.17, 47.23, 31.63) mm, rotated rx 180 ry 0 rz 180 deg; joints [-18.817, 18.265, 45.278, 37.411, 32.068, -32.949]
  MoveL 1201 to (240.17, 47.23, 31.63) mm, rotated rx 180 ry 0 rz 180 deg; joints [-18.817, 18.265, 45.278, 37.411, 32.068, -32.949]
  Call Extruder(202.27340)
  MoveL 1202 to (240.22, 47.43, 31.63) mm, rotated rx 180 ry 0 rz 180 deg; joints [-18.837, 18.289, 45.245, 37.434, 32.086, -32.966]
  MoveL 1203 to (240.22, 47.43, 31.63) mm, rotated rx 180 ry 0 rz 180 deg; joints [-18.837, 18.289, 45.245, 37.434, 32.086, -32.966]
  Call Extruder(202.41068)
  MoveL 1204 to (240.27, 47.68, 31.63) mm, rotated rx 180 ry 0 rz 180 deg; joints [-18.862, 18.318, 45.206, 37.463, 32.108, -32.987]
  MoveL 1205 to (240.27, 47.68, 31.63) mm, rotated rx 180 ry 0 rz 180 deg; joints [-18.862, 18.318, 45.206, 37.463, 32.108, -32.987]
  Call Extruder(202.54735)
  MoveL 1206 to (240.32, 47.93, 31.63) mm, rotated rx 180 ry 0 rz 180 deg; joints [-18.887, 18.347, 45.167, 37.492, 32.129, -33.009]
  MoveL 1207 to (240.32, 47.93, 31.63) mm, rotated rx 180 ry 0 rz 180 deg; joints [-18.887, 18.347, 45.167, 37.492, 32.129, -33.009]
  Call Extruder(202.68342)
  MoveL 1208 to (240.37, 48.18, 31.63) mm, rotated rx 180 ry 0 rz 180 deg; joints [-18.911, 18.376, 45.128, 37.52, 32.151, -33.029]
  MoveL 1209 to (240.37, 48.18, 31.63) mm, rotated rx 180 ry 0 rz 180 deg; joints [-18.911, 18.376, 45.128, 37.52, 32.151, -33.029]
  Call Extruder(202.81887)
  MoveL 1210 to (240.42, 48.43, 31.63) mm, rotated rx 180 ry 0 rz 180 deg; joints [-18.936, 18.404, 45.089, 37.549, 32.172, -33.05]
  MoveL 1211 to (240.42, 48.43, 31.63) mm, rotated rx 180 ry 0 rz 180 deg; joints [-18.936, 18.404, 45.089, 37.549, 32.172, -33.05]
  Call Extruder(202.95371)
  MoveL 1212 to (240.47, 48.68, 31.63) mm, rotated rx 180 ry 0 rz 180 deg; joints [-18.96, 18.433, 45.049, 37.578, 32.194, -33.071]
  MoveL 1213 to (240.47, 48.68, 31.63) mm, rotated rx 180 ry 0 rz 180 deg; joints [-18.96, 18.433, 45.049, 37.578, 32.194, -33.071]
  Call Extruder(203.08794)
  MoveL 1214 to (240.52, 48.93, 31.63) mm, rotated rx 180 ry 0 rz 180 deg; joints [-18.985, 18.463, 45.01, 37.606, 32.216, -33.092]
  MoveL 1215 to (240.52, 48.93, 31.63) mm, rotated rx 180 ry 0 rz 180 deg; joints [-18.985, 18.463, 45.01, 37.606, 32.216, -33.092]
  Call Extruder(203.22156)
  MoveL 1216 to (240.57, 49.17, 31.63) mm, rotated rx 180 ry 0 rz 180 deg; joints [-19.009, 18.491, 44.97, 37.635, 32.237, -33.113]
  MoveL 1217 to (240.57, 49.17, 31.63) mm, rotated rx 180 ry 0 rz 180 deg; joints [-19.009, 18.491, 44.97, 37.635, 32.237, -33.113]
  Call Extruder(203.38367)
  MoveL 1218 to (240.61, 49.48, 31.63) mm, rotated rx -180 ry 0 rz 180 deg; joints [-19.04, 18.525, 44.925, 37.671, 32.263, -33.139]
  MoveL 1219 to (240.61, 49.48, 31.63) mm, rotated rx -180 ry 0 rz 180 deg; joints [-19.04, 18.525, 44.925, 37.671, 32.263, -33.139]
  Call Extruder(203.54505)
  MoveL 1220 to (240.66, 49.79, 31.63) mm, rotated rx -180 ry 0 rz 180 deg; joints [-19.07, 18.558, 44.88, 37.707, 32.289, -33.166]
  MoveL 1221 to (240.66, 49.79, 31.63) mm, rotated rx -180 ry 0 rz 180 deg; joints [-19.07, 18.558, 44.88, 37.707, 32.289, -33.166]
  Call Extruder(203.70571)
  MoveL 1222 to (240.71, 50.09, 31.63) mm, rotated rx 180 ry 0 rz -180 deg; joints [-19.101, 18.591, 44.835, 37.743, 32.316, -33.193]
  MoveL 1223 to (240.71, 50.09, 31.63) mm, rotated rx 180 ry 0 rz -180 deg; joints [-19.101, 18.591, 44.835, 37.743, 32.316, -33.193]
  Call Extruder(203.86563)
  MoveL 1224 to (240.76, 50.4, 31.63) mm, rotated rx 180 ry 0 rz 180 deg; joints [-19.131, 18.624, 44.79, 37.779, 32.342, -33.219]
  MoveL 1225 to (240.76, 50.4, 31.63) mm, rotated rx 180 ry 0 rz 180 deg; joints [-19.131, 18.624, 44.79, 37.779, 32.342, -33.219]
  Call Extruder(204.02483)
  MoveL 1226 to (240.81, 50.7, 31.63) mm, rotated rx 180 ry 0 rz 180 deg; joints [-19.162, 18.658, 44.744, 37.815, 32.368, -33.246]
  MoveL 1227 to (240.81, 50.7, 31.63) mm, rotated rx 180 ry 0 rz 180 deg; joints [-19.162, 18.658, 44.744, 37.815, 32.368, -33.246]
  Call Extruder(204.18330)
  MoveL 1228 to (240.86, 51.01, 31.63) mm, rotated rx -180 ry 0 rz 180 deg; joints [-19.192, 18.691, 44.699, 37.851, 32.394, -33.272]
  MoveL 1229 to (240.86, 51.01, 31.63) mm, rotated rx -180 ry 0 rz 180 deg; joints [-19.192, 18.691, 44.699, 37.851, 32.394, -33.272]
  Call Extruder(204.38218)
  MoveL 1230 to (240.9, 51.4, 31.63) mm, rotated rx 180 ry 0 rz 180 deg; joints [-19.231, 18.73, 44.645, 37.898, 32.427, -33.307]
  MoveL 1231 to (240.9, 51.4, 31.63) mm, rotated rx 180 ry 0 rz 180 deg; joints [-19.231, 18.73, 44.645, 37.898, 32.427, -33.307]
  Call Extruder(204.58019)
  MoveL 1232 to (240.95, 51.78, 31.63) mm, rotated rx -180 ry 0 rz 180 deg; joints [-19.27, 18.769, 44.592, 37.945, 32.46, -33.342]
  MoveL 1233 to (240.95, 51.78, 31.63) mm, rotated rx -180 ry 0 rz 180 deg; joints [-19.27, 18.769, 44.592, 37.945, 32.46, -33.342]
  Call Extruder(204.77733)
  MoveL 1234 to (240.99, 52.17, 31.63) mm, rotated rx -180 ry 0 rz -180 deg; joints [-19.309, 18.809, 44.538, 37.992, 32.493, -33.377]
  MoveL 1235 to (240.99, 52.17, 31.63) mm, rotated rx -180 ry 0 rz -180 deg; joints [-19.309, 18.809, 44.538, 37.992, 32.493, -33.377]
  Call Extruder(204.97360)
  MoveL 1236 to (241.04, 52.56, 31.63) mm, rotated rx 180 ry 0 rz 180 deg; joints [-19.348, 18.848, 44.484, 38.039, 32.525, -33.411]
  MoveL 1237 to (241.04, 52.56, 31.63) mm, rotated rx 180 ry 0 rz 180 deg; joints [-19.348, 18.848, 44.484, 38.039, 32.525, -33.411]
  Call Extruder(205.21931)
  MoveL 1238 to (241.09, 53.05, 31.63) mm, rotated rx -180 ry 0 rz 180 deg; joints [-19.398, 18.895, 44.42, 38.099, 32.566, -33.456]
  MoveL 1239 to (241.09, 53.05, 31.63) mm, rotated rx -180 ry 0 rz 180 deg; joints [-19.398, 18.895, 44.42, 38.099, 32.566, -33.456]
  Call Extruder(205.51408)
  MoveL 1240 to (241.13, 53.64, 31.63) mm, rotated rx -180 ry 0 rz 180 deg; joints [-19.458, 18.951, 44.344, 38.173, 32.616, -33.512]
  MoveL 1241 to (241.13, 53.64, 31.63) mm, rotated rx -180 ry 0 rz 180 deg; joints [-19.458, 18.951, 44.344, 38.173, 32.616, -33.512]
  Call Extruder(205.80752)
  MoveL 1242 to (241.18, 54.23, 31.63) mm, rotated rx -180 ry 0 rz 180 deg; joints [-19.518, 19.006, 44.268, 38.246, 32.665, -33.566]
  MoveL 1243 to (241.18, 54.23, 31.63) mm, rotated rx -180 ry 0 rz 180 deg; joints [-19.518, 19.006, 44.268, 38.246, 32.665, -33.566]
  Call Extruder(206.24086)
  MoveL 1244 to (241.23, 55.1, 31.63) mm, rotated rx -180 ry 0 rz -180 deg; joints [-19.608, 19.084, 44.161, 38.357, 32.737, -33.65]
  MoveL 1245 to (241.23, 55.1, 31.63) mm, rotated rx -180 ry 0 rz -180 deg; joints [-19.608, 19.084, 44.161, 38.357, 32.737, -33.65]
  Call Extruder(206.81303)
  MoveL 1246 to (241.27, 56.27, 31.63) mm, rotated rx 180 ry 0 rz 180 deg; joints [-19.728, 19.185, 44.023, 38.505, 32.833, -33.762]
  MoveL 1247 to (241.27, 56.27, 31.63) mm, rotated rx 180 ry 0 rz 180 deg; joints [-19.728, 19.185, 44.023, 38.505, 32.833, -33.762]
  Call Extruder(207.24073)
  MoveL 1248 to (241.29, 57.14, 31.63) mm, rotated rx 180 ry 0 rz 180 deg; joints [-19.819, 19.257, 43.923, 38.617, 32.905, -33.847]
  Call Extruder(249.23436)
  MoveL 1249 to (241.29, 142.86, 31.63) mm, rotated rx 180 ry 0 rz 180 deg; joints [-28.232, 29.39, 28.869, 45.584, 41.473, -37.405]
  MoveL 1250 to (241.29, 142.86, 31.63) mm, rotated rx 180 ry 0 rz 180 deg; joints [-28.232, 29.39, 28.869, 45.584, 41.473, -37.405]
  Call Extruder(249.94981)
  MoveL 1251 to (241.25, 144.32, 31.63) mm, rotated rx 180 ry 0 rz 180 deg; joints [-28.367, 29.655, 28.443, 45.616, 41.667, -37.353]
  MoveL 1252 to (241.25, 144.32, 31.63) mm, rotated rx 180 ry 0 rz 180 deg; joints [-28.367, 29.655, 28.443, 45.616, 41.667, -37.353]
  Call Extruder(250.52455)
  MoveL 1253 to (241.2, 145.48, 31.63) mm, rotated rx 180 ry 0 rz 180 deg; joints [-28.475, 29.867, 28.102, 45.642, 41.824, -37.311]
  MoveL 1254 to (241.2, 145.48, 31.63) mm, rotated rx 180 ry 0 rz 180 deg; joints [-28.475, 29.867, 28.102, 45.642, 41.824, -37.311]
  Call Extruder(250.81799)
  MoveL 1255 to (241.15, 146.07, 31.63) mm, rotated rx 180 ry 0 rz 180 deg; joints [-28.531, 29.967, 27.94, 45.659, 41.901, -37.294]
  MoveL 1256 to (241.15, 146.07, 31.63) mm, rotated rx 180 ry 0 rz 180 deg; joints [-28.531, 29.967, 27.94, 45.659, 41.901, -37.294]
  Call Extruder(251.11276)
  MoveL 1257 to (241.11, 146.66, 31.63) mm, rotated rx 180 ry 0 rz 180 deg; joints [-28.587, 30.069, 27.775, 45.676, 41.979, -37.276]
  MoveL 1258 to (241.11, 146.66, 31.63) mm, rotated rx 180 ry 0 rz 180 deg; joints [-28.587, 30.069, 27.775, 45.676, 41.979, -37.276]
  Call Extruder(251.40887)
  MoveL 1259 to (241.06, 147.25, 31.63) mm, rotated rx -180 ry 0 rz 180 deg; joints [-28.643, 30.172, 27.608, 45.692, 42.057, -37.257]
  MoveL 1260 to (241.06, 147.25, 31.63) mm, rotated rx -180 ry 0 rz 180 deg; joints [-28.643, 30.172, 27.608, 45.692, 42.057, -37.257]
  Call Extruder(251.60514)
  MoveL 1261 to (241.02, 147.64, 31.63) mm, rotated rx -180 ry 0 rz -180 deg; joints [-28.681, 30.235, 27.506, 45.705, 42.107, -37.248]
  MoveL 1262 to (241.02, 147.64, 31.63) mm, rotated rx -180 ry 0 rz -180 deg; joints [-28.681, 30.235, 27.506, 45.705, 42.107, -37.248]
  Call Extruder(251.80228)
  MoveL 1263 to (240.97, 148.02, 31.63) mm, rotated rx 180 ry 0 rz 180 deg; joints [-28.718, 30.298, 27.403, 45.718, 42.158, -37.239]
  MoveL 1264 to (240.97, 148.02, 31.63) mm, rotated rx 180 ry 0 rz 180 deg; joints [-28.718, 30.298, 27.403, 45.718, 42.158, -37.239]
  Call Extruder(252.00029)
  MoveL 1265 to (240.92, 148.41, 31.63) mm, rotated rx 180 ry 0 rz 180 deg; joints [-28.756, 30.361, 27.3, 45.731, 42.208, -37.23]
  MoveL 1266 to (240.92, 148.41, 31.63) mm, rotated rx 180 ry 0 rz 180 deg; joints [-28.756, 30.361, 27.3, 45.731, 42.208, -37.23]
  Call Extruder(252.19916)
  MoveL 1267 to (240.88, 148.8, 31.63) mm, rotated rx -180 ry 0 rz -180 deg; joints [-28.793, 30.425, 27.196, 45.744, 42.259, -37.22]
  MoveL 1268 to (240.88, 148.8, 31.63) mm, rotated rx -180 ry 0 rz -180 deg; joints [-28.793, 30.425, 27.196, 45.744, 42.259, -37.22]
  Call Extruder(252.37825)
  MoveL 1269 to (240.83, 149.14, 31.63) mm, rotated rx -180 ry 0 rz 180 deg; joints [-28.827, 30.481, 27.106, 45.756, 42.304, -37.212]
  MoveL 1270 to (240.83, 149.14, 31.63) mm, rotated rx -180 ry 0 rz 180 deg; joints [-28.827, 30.481, 27.106, 45.756, 42.304, -37.212]
  Call Extruder(252.53744)
  MoveL 1271 to (240.78, 149.45, 31.63) mm, rotated rx 180 ry 0 rz -180 deg; joints [-28.857, 30.527, 27.03, 45.769, 42.342, -37.208]
  MoveL 1272 to (240.78, 149.45, 31.63) mm, rotated rx 180 ry 0 rz -180 deg; joints [-28.857, 30.527, 27.03, 45.769, 42.342, -37.208]
  Call Extruder(252.69737)
  MoveL 1273 to (240.73, 149.76, 31.63) mm, rotated rx 180 ry 0 rz -180 deg; joints [-28.887, 30.574, 26.954, 45.781, 42.381, -37.202]
  MoveL 1274 to (240.73, 149.76, 31.63) mm, rotated rx 180 ry 0 rz -180 deg; joints [-28.887, 30.574, 26.954, 45.781, 42.381, -37.202]
  Call Extruder(252.85802)
  MoveL 1275 to (240.69, 150.06, 31.63) mm, rotated rx -180 ry 0 rz 180 deg; joints [-28.917, 30.621, 26.877, 45.794, 42.42, -37.197]
  MoveL 1276 to (240.69, 150.06, 31.63) mm, rotated rx -180 ry 0 rz 180 deg; joints [-28.917, 30.621, 26.877, 45.794, 42.42, -37.197]
  Call Extruder(253.01940)
  MoveL 1277 to (240.64, 150.37, 31.63) mm, rotated rx -180 ry 0 rz 180 deg; joints [-28.947, 30.668, 26.8, 45.805, 42.459, -37.191]
  MoveL 1278 to (240.64, 150.37, 31.63) mm, rotated rx -180 ry 0 rz 180 deg; joints [-28.947, 30.668, 26.8, 45.805, 42.459, -37.191]
  Call Extruder(253.18150)
  MoveL 1279 to (240.59, 150.67, 31.63) mm, rotated rx 180 ry 0 rz 180 deg; joints [-28.978, 30.716, 26.722, 45.817, 42.498, -37.185]
  MoveL 1280 to (240.59, 150.67, 31.63) mm, rotated rx 180 ry 0 rz 180 deg; joints [-28.978, 30.716, 26.722, 45.817, 42.498, -37.185]
  Call Extruder(253.32971)
  MoveL 1281 to (240.54, 150.95, 31.63) mm, rotated rx 180 ry 0 rz 180 deg; joints [-29.005, 30.757, 26.654, 45.829, 42.533, -37.181]
  MoveL 1282 to (240.54, 150.95, 31.63) mm, rotated rx 180 ry 0 rz 180 deg; joints [-29.005, 30.757, 26.654, 45.829, 42.533, -37.181]
  Call Extruder(253.46394)
  MoveL 1283 to (240.49, 151.2, 31.63) mm, rotated rx 180 ry 0 rz 180 deg; joints [-29.03, 30.793, 26.596, 45.841, 42.564, -37.179]
  MoveL 1284 to (240.49, 151.2, 31.63) mm, rotated rx 180 ry 0 rz 180 deg; joints [-29.03, 30.793, 26.596, 45.841, 42.564, -37.179]
  Call Extruder(253.59878)
  MoveL 1285 to (240.44, 151.45, 31.63) mm, rotated rx 180 ry 0 rz 180 deg; joints [-29.055, 30.828, 26.538, 45.853, 42.595, -37.177]
  MoveL 1286 to (240.44, 151.45, 31.63) mm, rotated rx 180 ry 0 rz 180 deg; joints [-29.055, 30.828, 26.538, 45.853, 42.595, -37.177]
  Call Extruder(253.73424)
  MoveL 1287 to (240.39, 151.7, 31.63) mm, rotated rx -180 ry 0 rz 180 deg; joints [-29.08, 30.864, 26.48, 45.864, 42.626, -37.174]
  MoveL 1288 to (240.39, 151.7, 31.63) mm, rotated rx -180 ry 0 rz 180 deg; joints [-29.08, 30.864, 26.48, 45.864, 42.626, -37.174]
  Call Extruder(253.87030)
  MoveL 1289 to (240.34, 151.95, 31.63) mm, rotated rx -180 ry 0 rz 180 deg; joints [-29.105, 30.899, 26.421, 45.876, 42.657, -37.171]
  MoveL 1290 to (240.34, 151.95, 31.63) mm, rotated rx -180 ry 0 rz 180 deg; joints [-29.105, 30.899, 26.421, 45.876, 42.657, -37.171]
  Call Extruder(254.00697)
  MoveL 1291 to (240.29, 152.2, 31.63) mm, rotated rx 180 ry 0 rz 180 deg; joints [-29.13, 30.936, 26.362, 45.887, 42.688, -37.168]
  MoveL 1292 to (240.29, 152.2, 31.63) mm, rotated rx 180 ry 0 rz 180 deg; joints [-29.13, 30.936, 26.362, 45.887, 42.688, -37.168]
  Call Extruder(254.14425)
  MoveL 1293 to (240.24, 152.45, 31.63) mm, rotated rx 180 ry 0 rz 180 deg; joints [-29.155, 30.972, 26.303, 45.898, 42.72, -37.166]
  MoveL 1294 to (240.24, 152.45, 31.63) mm, rotated rx 180 ry 0 rz 180 deg; joints [-29.155, 30.972, 26.303, 45.898, 42.72, -37.166]
  Call Extruder(254.26992)
  MoveL 1295 to (240.2, 152.67, 31.63) mm, rotated rx 180 ry 0 rz -180 deg; joints [-29.178, 31.004, 26.25, 45.909, 42.748, -37.163]
  MoveL 1296 to (240.2, 152.67, 31.63) mm, rotated rx 180 ry 0 rz -180 deg; joints [-29.178, 31.004, 26.25, 45.909, 42.748, -37.163]
  Call Extruder(254.38384)
  MoveL 1297 to (240.15, 152.88, 31.63) mm, rotated rx 180 ry 0 rz 180 deg; joints [-29.198, 31.032, 26.203, 45.919, 42.773, -37.162]
  MoveL 1298 to (240.15, 152.88, 31.63) mm, rotated rx 180 ry 0 rz 180 deg; joints [-29.198, 31.032, 26.203, 45.919, 42.773, -37.162]
  Call Extruder(254.49822)
  MoveL 1299 to (240.11, 153.08, 31.63) mm, rotated rx 180 ry 0 rz 180 deg; joints [-29.219, 31.061, 26.156, 45.929, 42.798, -37.16]
  MoveL 1300 to (240.11, 153.08, 31.63) mm, rotated rx 180 ry 0 rz 180 deg; joints [-29.219, 31.061, 26.156, 45.929, 42.798, -37.16]
  Call Extruder(254.61305)
  MoveL 1301 to (240.06, 153.28, 31.63) mm, rotated rx 180 ry 0 rz -180 deg; joints [-29.24, 31.089, 26.11, 45.939, 42.823, -37.158]
  MoveL 1302 to (240.06, 153.28, 31.63) mm, rotated rx 180 ry 0 rz -180 deg; joints [-29.24, 31.089, 26.11, 45.939, 42.823, -37.158]
  Call Extruder(254.72833)
  MoveL 1303 to (240.02, 153.49, 31.63) mm, rotated rx -180 ry 0 rz 180 deg; joints [-29.26, 31.117, 26.063, 45.949, 42.849, -37.157]
  MoveL 1304 to (240.02, 153.49, 31.63) mm, rotated rx -180 ry 0 rz 180 deg; joints [-29.26, 31.117, 26.063, 45.949, 42.849, -37.157]
  Call Extruder(254.85771)
  MoveL 1305 to (239.95, 153.71, 31.63) mm, rotated rx 180 ry 0 rz -180 deg; joints [-29.284, 31.141, 26.023, 45.965, 42.874, -37.161]
  MoveL 1306 to (239.95, 153.71, 31.63) mm, rotated rx 180 ry 0 rz -180 deg; joints [-29.284, 31.141, 26.023, 45.965, 42.874, -37.161]
  Call Extruder(254.98765)
  MoveL 1307 to (239.88, 153.94, 31.63) mm, rotated rx 180 ry 0 rz -180 deg; joints [-29.307, 31.165, 25.984, 45.98, 42.899, -37.164]
  MoveL 1308 to (239.88, 153.94, 31.63) mm, rotated rx 180 ry 0 rz -180 deg; joints [-29.307, 31.165, 25.984, 45.98, 42.899, -37.164]
  Call Extruder(255.11816)
  MoveL 1309 to (239.82, 154.16, 31.63) mm, rotated rx 180 ry 0 rz 180 deg; joints [-29.331, 31.189, 25.944, 45.996, 42.924, -37.168]
  MoveL 1310 to (239.82, 154.16, 31.63) mm, rotated rx 180 ry 0 rz 180 deg; joints [-29.331, 31.189, 25.944, 45.996, 42.924, -37.168]
  Call Extruder(255.24923)
  MoveL 1311 to (239.75, 154.38, 31.63) mm, rotated rx -180 ry 0 rz 180 deg; joints [-29.354, 31.213, 25.904, 46.011, 42.949, -37.172]
  MoveL 1312 to (239.75, 154.38, 31.63) mm, rotated rx -180 ry 0 rz 180 deg; joints [-29.354, 31.213, 25.904, 46.011, 42.949, -37.172]
  Call Extruder(255.37087)
  MoveL 1313 to (239.68, 154.59, 31.63) mm, rotated rx -180 ry 0 rz -180 deg; joints [-29.376, 31.235, 25.87, 46.026, 42.972, -37.176]
  MoveL 1314 to (239.68, 154.59, 31.63) mm, rotated rx -180 ry 0 rz -180 deg; joints [-29.376, 31.235, 25.87, 46.026, 42.972, -37.176]
  Call Extruder(255.48300)
  MoveL 1315 to (239.62, 154.78, 31.63) mm, rotated rx 180 ry 0 rz 180 deg; joints [-29.396, 31.253, 25.839, 46.04, 42.992, -37.18]
  MoveL 1316 to (239.62, 154.78, 31.63) mm, rotated rx 180 ry 0 rz 180 deg; joints [-29.396, 31.253, 25.839, 46.04, 42.992, -37.18]
  Call Extruder(255.59556)
  MoveL 1317 to (239.56, 154.97, 31.63) mm, rotated rx -180 ry 0 rz 180 deg; joints [-29.416, 31.272, 25.807, 46.054, 43.013, -37.184]
  MoveL 1318 to (239.56, 154.97, 31.63) mm, rotated rx -180 ry 0 rz 180 deg; joints [-29.416, 31.272, 25.807, 46.054, 43.013, -37.184]
  Call Extruder(255.70858)
  MoveL 1319 to (239.5, 155.15, 31.63) mm, rotated rx -180 ry 0 rz 180 deg; joints [-29.436, 31.291, 25.776, 46.068, 43.033, -37.188]
  MoveL 1320 to (239.5, 155.15, 31.63) mm, rotated rx -180 ry 0 rz 180 deg; joints [-29.436, 31.291, 25.776, 46.068, 43.033, -37.188]
  Call Extruder(255.82203)
  MoveL 1321 to (239.44, 155.34, 31.63) mm, rotated rx -180 ry 0 rz 180 deg; joints [-29.456, 31.31, 25.745, 46.082, 43.054, -37.193]
  MoveL 1322 to (239.44, 155.34, 31.63) mm, rotated rx -180 ry 0 rz 180 deg; joints [-29.456, 31.31, 25.745, 46.082, 43.054, -37.193]
  Call Extruder(255.96967)
  MoveL 1323 to (239.35, 155.58, 31.63) mm, rotated rx 180 ry 0 rz 180 deg; joints [-29.483, 31.328, 25.714, 46.103, 43.078, -37.202]
  MoveL 1324 to (239.35, 155.58, 31.63) mm, rotated rx 180 ry 0 rz 180 deg; joints [-29.483, 31.328, 25.714, 46.103, 43.078, -37.202]
  Call Extruder(256.15201)
  MoveL 1325 to (239.22, 155.87, 31.63) mm, rotated rx 180 ry 0 rz 180 deg; joints [-29.515, 31.347, 25.684, 46.131, 43.106, -37.217]
  MoveL 1326 to (239.22, 155.87, 31.63) mm, rotated rx 180 ry 0 rz 180 deg; joints [-29.515, 31.347, 25.684, 46.131, 43.106, -37.217]
  Call Extruder(256.33510)
  MoveL 1327 to (239.11, 156.17, 31.63) mm, rotated rx 180 ry 0 rz 180 deg; joints [-29.547, 31.366, 25.652, 46.159, 43.134, -37.231]
  MoveL 1328 to (239.11, 156.17, 31.63) mm, rotated rx 180 ry 0 rz 180 deg; joints [-29.547, 31.366, 25.652, 46.159, 43.134, -37.231]
  Call Extruder(256.49281)
  MoveL 1329 to (239, 156.42, 31.63) mm, rotated rx 180 ry 0 rz 180 deg; joints [-29.575, 31.381, 25.628, 46.184, 43.158, -37.245]
  MoveL 1330 to (239, 156.42, 31.63) mm, rotated rx 180 ry 0 rz 180 deg; joints [-29.575, 31.381, 25.628, 46.184, 43.158, -37.245]
  Call Extruder(256.65113)
  MoveL 1331 to (238.89, 156.66, 31.63) mm, rotated rx -180 ry 0 rz 180 deg; joints [-29.603, 31.395, 25.604, 46.209, 43.181, -37.258]
  MoveL 1332 to (238.89, 156.66, 31.63) mm, rotated rx -180 ry 0 rz 180 deg; joints [-29.603, 31.395, 25.604, 46.209, 43.181, -37.258]
  Call Extruder(256.83316)
  MoveL 1333 to (238.75, 156.94, 31.63) mm, rotated rx 180 ry 0 rz -180 deg; joints [-29.635, 31.402, 25.593, 46.243, 43.203, -37.281]
  MoveL 1334 to (238.75, 156.94, 31.63) mm, rotated rx 180 ry 0 rz -180 deg; joints [-29.635, 31.402, 25.593, 46.243, 43.203, -37.281]
  Call Extruder(257.03972)
  MoveL 1335 to (238.57, 157.25, 31.63) mm, rotated rx 180 ry 0 rz 180 deg; joints [-29.671, 31.401, 25.595, 46.286, 43.225, -37.312]
  MoveL 1336 to (238.57, 157.25, 31.63) mm, rotated rx 180 ry 0 rz 180 deg; joints [-29.671, 31.401, 25.595, 46.286, 43.225, -37.312]
  Call Extruder(257.24706)
  MoveL 1337 to (238.4, 157.55, 31.63) mm, rotated rx -180 ry 0 rz 180 deg; joints [-29.707, 31.4, 25.596, 46.328, 43.247, -37.343]
  MoveL 1338 to (238.4, 157.55, 31.63) mm, rotated rx -180 ry 0 rz 180 deg; joints [-29.707, 31.4, 25.596, 46.328, 43.247, -37.343]
  Call Extruder(257.45518)
  MoveL 1339 to (238.22, 157.85, 31.63) mm, rotated rx 180 ry 0 rz 180 deg; joints [-29.743, 31.399, 25.598, 46.371, 43.268, -37.375]
  MoveL 1340 to (238.22, 157.85, 31.63) mm, rotated rx 180 ry 0 rz 180 deg; joints [-29.743, 31.399, 25.598, 46.371, 43.268, -37.375]
  Call Extruder(257.57289)
  MoveL 1341 to (238.12, 158.02, 31.63) mm, rotated rx -180 ry 0 rz 180 deg; joints [-29.764, 31.399, 25.598, 46.395, 43.28, -37.392]
  MoveL 1342 to (238.12, 158.02, 31.63) mm, rotated rx -180 ry 0 rz 180 deg; joints [-29.764, 31.399, 25.598, 46.395, 43.28, -37.392]
  Call Extruder(257.90571)
  MoveL 1343 to (237.79, 158.48, 31.63) mm, rotated rx 180 ry 0 rz 180 deg; joints [-29.821, 31.369, 25.647, 46.476, 43.302, -37.461]
  MoveL 1344 to (237.79, 158.48, 31.63) mm, rotated rx 180 ry 0 rz 180 deg; joints [-29.821, 31.369, 25.647, 46.476, 43.302, -37.461]
  Call Extruder(258.23971)
  MoveL 1345 to (237.47, 158.93, 31.63) mm, rotated rx 180 ry 0 rz 180 deg; joints [-29.878, 31.34, 25.695, 46.556, 43.323, -37.529]
  MoveL 1346 to (237.47, 158.93, 31.63) mm, rotated rx 180 ry 0 rz 180 deg; joints [-29.878, 31.34, 25.695, 46.556, 43.323, -37.529]
  Call Extruder(258.40729)
  MoveL 1347 to (237.3, 159.15, 31.63) mm, rotated rx -180 ry 0 rz 180 deg; joints [-29.907, 31.326, 25.719, 46.597, 43.335, -37.563]
  Call Extruder(259.23663)
  MoveL 1348 to (236.39, 160.19, 31.63) mm, rotated rx 180 ry 0 rz 180 deg; joints [-30.046, 31.196, 25.934, 46.823, 43.362, -37.77]
  Call Extruder(259.86767)
  MoveL 1349 to (235.6, 160.89, 31.63) mm, rotated rx 180 ry 0 rz 180 deg; joints [-30.149, 31.04, 26.19, 47.019, 43.356, -37.963]
